    PRINTER_STATES.DataReady :                        // Wait for command to begin printing
                                                    IF NOT printerDataReady THEN
														state := PRINTER_STATES.Idle;
													END_IF
													IF _mode = DEVICE_MODES.Auto AND _amPrintNow THEN
                                                        state := PRINTER_STATES.BeginPrintCycle;
                                                        _amPrintNow := FALSE;
														printHeadDebounce.IN := TRUE;
                                                        oLowerPrintHead := TRUE;
                                                        oRunPrinterRibbonUnwindMotor := TRUE;
														//oPrinterStartPrint := TRUE;
                                                    END_IF                                    
            
    
    PRINTER_STATES.BeginPrintCycle :                // Start printing
                                                    
                                                    
                                                    IF _amSendPrintSignal THEN
                                                        oPrinterStartPrint := TRUE;
														
                                                        state := PRINTER_STATES.Printing;
                                                        printHeadDebounce.IN := FALSE;
                                                        _amSendPrintSignal := FALSE;
                                                    END_IF                                                    
                                        
    
    PRINTER_STATES.FeedAtPrintSpeed :                //

                                                    
                                                                                                
                                        
    PRINTER_STATES.Printing :                        //While printing, wait for End of Print signal
													printerRibbonMovingTimer1.IN := ribbonEncoderPulse;
													printerRibbonMovingTimer2.IN := NOT ribbonEncoderPulse;
                                                    IF endOfPrintONS.Q OR printerRibbonMovingTimer1.Q OR printerRibbonMovingTimer2.Q THEN
                                                        oPrinterStartPrint := FALSE;
                                                        oLowerPrintHead := FALSE;
														IF printerRibbonMovingTimer1.Q OR printerRibbonMovingTimer2.Q THEN
															ribbonFault.Trigger();
														END_IF
														printerRibbonMovingTimer1.IN := FALSE;
														printerRibbonMovingTimer2.IN := FALSE;
														 
                                                        //oRunPrinterRibbonUnwindMotor := FALSE;
                                                        state := PRINTER_STATES.DonePrinting;    
                                                    END_IF
                                        
    PRINTER_STATES.DonePrinting :                    //Done printing, feed a little more through
                                                    IF _mode = DEVICE_MODES.Auto AND _amGoToIdle THEN
                                                        oRunPrinterRibbonUnwindMotor := FALSE;
                                                        state := PRINTER_STATES.Idle;
                                                        _amGoToIdle := FALSE;
														HMIData.printerCycles.Increment();
														HMIData.printHeadClean.Increment();
                                                        Globals.printerCycleCounts := Globals.printerCycleCounts + 1;
                                                    END_IF
        
    PRINTER_STATES.FeedThrough :                        
                                        
    PRINTER_STATES.Ready :                        
                                        
    PRINTER_STATES.Fault :                        
                                        
END_CASE

METHOD AutoSendPrintSignal
VAR_INPUT
END_VAR
_amSendPrintSignal := TRUE;
END_METHOD

METHOD AutoPrintNow
VAR_INPUT
END_VAR
_amPrintNow := TRUE;
END_METHOD

METHOD AutoAckPrintDone
VAR_INPUT
END_VAR
_amGoToIdle := TRUE;
END_METHOD

PROPERTY Ready : BOOL
SET
_ready := Ready;
END_SET
GET
Ready := _ready;
END_GET
END_PROPERTY

PROPERTY Mode : DEVICE_MODES
SET
_mode := Mode;
END_SET
GET
Mode := _mode;
END_GET
END_PROPERTY

END_FUNCTION_BLOCK

// Device/Application/FBs/Components/MonostableMultivibratorFB
FUNCTION_BLOCK MonostableMultivibratorFB EXTENDS BaseComponentFB
VAR_INPUT
END_VAR
VAR_OUTPUT
	Q : BOOL;   // Output pulse
END_VAR
VAR
	_trigger : BOOL;
	_dwellTimeInMS : UINT := 80; 	// Pulse Dwell in mS 
	_delayTimeInMS : UINT; 			// Delay before Pulse in mS
	_manualOn : BOOL;
	_manualOff : BOOL;
	active : BOOL;
	dwellTimer : Standard.TON;
	delayTimer : Standard.TON;
END_VAR


// HPA is on for only as long as its setpoint.

delayTimer(IN := _trigger AND NOT dwellTimer.Q, PT := UINT_TO_TIME(_delayTimeInMS));
dwellTimer(IN := delayTimer.Q AND NOT dwellTimer.Q, PT := UINT_TO_TIME(_dwellTimeInMS));

Q:= delayTimer.Q OR _manualOn;

IF dwellTimer.Q OR _reset THEN
	active := FALSE;
	_trigger := FALSE;
	_manualOn := FALSE;
	_manualOff := FALSE;
END_IF

SUPER^();

PROPERTY DelaySetting : UINT
GET
DelaySetting := _delayTimeInMS;
END_GET
SET
_delayTimeInMS := DelaySetting;
END_SET
END_PROPERTY

METHOD Trigger
VAR_INPUT
END_VAR
_trigger := TRUE;
END_METHOD

METHOD ManualOn
VAR_INPUT
END_VAR
_manualOn := TRUE;
_manualOff := FALSE;
END_METHOD

METHOD ManualOff : BOOL
VAR_INPUT
END_VAR
_manualOn := FALSE;
_manualOff := TRUE;
END_METHOD

PROPERTY DwellSetting : UINT
SET
_dwellTimeInMS := DwellSetting;
END_SET
GET
DwellSetting := _dwellTimeInMS;
END_GET
END_PROPERTY

END_FUNCTION_BLOCK

// Device/Application/FBs/Components/DelayDwellFB/DelayDwellFB
FUNCTION_BLOCK DelayDwellFB EXTENDS BaseComponentFB
VAR_INPUT
END_VAR
VAR_OUTPUT
	Q : BOOL;   // Output pulse
END_VAR
VAR
	_trigger : BOOL;
	_dwellTimeInMS : DINT := 80; 	// Pulse Dwell in mS 
	_delayTimeInMS : DINT; 			// Delay before Pulse in mS
	_manualOn : BOOL;
	_manualOff : BOOL;
	active : BOOL;
	dwellTimer : Standard.TON;
	delayTimer : Standard.TON;
	state : DELAY_DWELL_STATES;
END_VAR

//    Function Block: DelayDwellFB
//    Description: On Trigger(), starts a delay then sets the Q output for a dwell time.  Each addition Trigger() resets the dwell timer.
//    Created by: Ben Hess
//    Created Date: February 20th, 2020

// Setup timers for reading offset and scanning distance
delayTimer(PT := UDINT_TO_TIME(_delayTimeInMS));
// If negative dwell time, run forever
IF _dwellTimeInMS < 0 THEN
	dwellTimer(PT := T#0MS);
ELSE
	dwellTimer(PT := UDINT_TO_TIME(_dwellTimeInMS));
END_IF

// Manual On/Off
IF _manualOff THEN
	THIS^.Reset();
	state := DELAY_DWELL_STATES.Idle;
ELSIF _manualOn THEN
	THIS^.Reset();
	Q := TRUE;
	state := DELAY_DWELL_STATES.Idle;
END_IF

CASE state OF
	DELAY_DWELL_STATES.Idle:  			//
										dwellTimer.IN := FALSE;
										delayTimer.IN := FALSE;
										
										IF _trigger THEN
											IF _delayTimeInMS <> 0 THEN
												state := DELAY_DWELL_STATES.Delay;
											ELSE
												state := DELAY_DWELL_STATES.Dwell;
											END_IF
											_trigger := FALSE;
										END_IF
	
	DELAY_DWELL_STATES.Delay: 			//
										delayTimer.IN := TRUE;
										IF delayTimer.Q THEN
											delayTimer.IN := FALSE;
											state := DELAY_DWELL_STATES.Dwell;
										END_IF
	
	DELAY_DWELL_STATES.Dwell: 			//
										Q := TRUE;
										IF _dwellTimeInMS >= 0 THEN
											dwellTimer.IN := TRUE;
											IF dwellTimer.Q THEN
												dwellTimer.IN := FALSE;
												Q := FALSE;
												state := DELAY_DWELL_STATES.Idle;
											END_IF
										END_IF
										IF _trigger THEN
											_trigger := FALSE;
											state := DELAY_DWELL_STATES.ResettingDwell;
										END_IF
										
	DELAY_DWELL_STATES.ResettingDwell: 	//
										dwellTimer.IN := FALSE;
										state := DELAY_DWELL_STATES.Dwell;
END_CASE

SUPER^();

METHOD Reset : BOOL
VAR_INPUT
END_VAR
active := FALSE;
_trigger := FALSE;
_manualOn := FALSE;
_manualOff := FALSE;
Q := FALSE;
state := DELAY_DWELL_STATES.Idle;
END_METHOD

METHOD ManualOff : BOOL
VAR_INPUT
END_VAR
_manualOn := FALSE;
_manualOff := TRUE;
END_METHOD

METHOD ManualOn
VAR_INPUT
END_VAR
_manualOn := TRUE;
_manualOff := FALSE;
END_METHOD

METHOD Trigger
VAR_INPUT
END_VAR
_trigger := TRUE;
END_METHOD

PROPERTY DwellSetting : DINT
GET
DwellSetting := _dwellTimeInMS;
END_GET
SET
_dwellTimeInMS := DwellSetting;
END_SET
END_PROPERTY

PROPERTY DelaySetting : DINT
SET
_delayTimeInMS := DelaySetting;
END_SET
GET
DelaySetting := _delayTimeInMS;
END_GET
END_PROPERTY

END_FUNCTION_BLOCK

// Device/Application/FBs/Components/BagOpenFingersWithSensorsFB
FUNCTION_BLOCK BagOpenFingersWithSensorsFB EXTENDS BagOpenFingersFB
VAR_INPUT
	rightFingerBagPresent : BOOL;
	leftFingerBagPreset : BOOL;
END_VAR
VAR_IN_OUT
	bagFailedToGrabBothFingersCount : UDINT; // Both Fingers failed to grab bag
	bagFailedToGrabRightFingerCount : UDINT; // Right Bag Open Finger Failed to Grab Bag
	bagFailedToGrabLeftFingerCount : UDINT; // Left Bag Open Finger Failed to Grab Bag
	successfulBagOpenCount : UDINT;			// Successful Bag Open Count
END_VAR
VAR_OUTPUT
	
END_VAR

SUPER^();

METHOD CheckIfBagGrabbed : BOOL
VAR_INPUT
	incrementCounters : BOOL; // IF TRUE Incerment bag counters, otherwise just return bag grabbed status
END_VAR
// Returns true if bag grab successful.  Also increments appropriate counters

{warning disable C0371}
// Checking the VAR_IN_OUT reference, leave the current method in case of invalid reference
IF NOT __ISVALIDREF(successfulBagOpenCount) 
	OR NOT __ISVALIDREF(bagFailedToGrabLeftFingerCount)
	OR NOT __ISVALIDREF(bagFailedToGrabRightFingerCount)
	OR NOT __ISVALIDREF(bagFailedToGrabBothFingersCount)
	THEN RETURN;    
END_IF

IF rightFingerBagPresent AND leftFingerBagPreset THEN
	IF incrementCounters THEN
		successfulBagOpenCount := successfulBagOpenCount +1;
	END_IF
	CheckIfBagGrabbed := TRUE;
ELSIF rightFingerBagPresent AND NOT leftFingerBagPreset THEN
	IF incrementCounters THEN
		bagFailedToGrabLeftFingerCount := bagFailedToGrabLeftFingerCount +1 ;
	END_IF
ELSIF NOT rightFingerBagPresent AND leftFingerBagPreset THEN
	IF incrementCounters THEN
		bagFailedToGrabRightFingerCount := bagFailedToGrabRightFingerCount + 1;
	END_IF
ELSE
	IF incrementCounters THEN
		bagFailedToGrabBothFingersCount := bagFailedToGrabBothFingersCount + 1;
	END_IF
END_IF
{warning restore C0371}
END_METHOD

END_FUNCTION_BLOCK

// Device/Application/FBs/Components/BagOpenFingersFB
FUNCTION_BLOCK BagOpenFingersFB EXTENDS BaseComponentFB
VAR_INPUT

END_VAR
VAR_IN_OUT

END_VAR
VAR_OUTPUT
    releaseOutput : BOOL;
	grabOutput : BOOL;
END_VAR
VAR
    _releaseCommand : BOOL;
    _grabCommand : BOOL;
END_VAR

SUPER^();
releaseOutput := _releaseCommand AND enable;
grabOutput := _grabCommand AND enable;

METHOD Release
VAR_INPUT
END_VAR
_releaseCommand := TRUE;
_grabCommand := FALSE;
END_METHOD

METHOD Grab
VAR_INPUT
END_VAR
_releaseCommand := FALSE;
_grabCommand := TRUE;
HMIData.bagOpenFingerCycles.Increment();
END_METHOD

END_FUNCTION_BLOCK

// Device/Application/FBs/Motors/Applied Motion/FB_AppliedMotionStepServoEIPPassthrough
FUNCTION_BLOCK FB_AppliedMotionStepServoEIPPassthrough EXTENDS FB_AppliedMotionStepServoEIPBase
VAR_INPUT
END_VAR
VAR_OUTPUT
END_VAR
VAR
	homingState : JAW_HOMING_STATES;
	homeRequiredONS : R_TRIG;
	timerHomeDelay : TON;
END_VAR

SUPER^();

METHOD HomeNow
_homeNow := TRUE;
END_METHOD

METHOD DoneClamping
VAR_INPUT
END_VAR
sclCommand := 16#434D; // CM Control Mode
parameter1 := 21;
															
commandSuccessful := FALSE;
commands.SendHostCommand := TRUE;
END_METHOD

METHOD AllowClamping
VAR_INPUT
END_VAR
sclCommand := 16#434D; // CM Control Mode
parameter1 := 1;
															
commandSuccessful := FALSE;
commands.SendHostCommand := TRUE;
END_METHOD

//{warning 'add method implementation '}
METHOD Stop
commandSuccessful := FALSE;
commands.StopCrash := TRUE;
END_METHOD

METHOD SetPositionLimit
VAR_INPUT
	positionLimit : DINT;
END_VAR
sclCommand := 16#5046; // PF (Position Fault)
parameter1 := positionLimit;
															
commandSuccessful := FALSE;
commands.SendHostCommand := TRUE;
END_METHOD

METHOD Execute
VAR_INPUT
END_VAR
SUPER^.Execute();
timerHomeDelay();
homeRequiredONS(CLK := homeRequiredIndication);

//IF _reset OR homeRequiredONS.Q THEN
IF _reset THEN
	homingState := JAW_HOMING_STATES.Idle;
	_homeNow := FALSE;
	timerHomeDelay.IN := FALSE;
END_IF

CASE homingState OF
	JAW_HOMING_STATES.Idle:						IF _homeNow THEN
													//IF NOT driveInputs[10].2 THEN
													//	homingState := JAW_HOMING_STATES.MoveForwardFromSensor;
													//ELSE 
														homingState := JAW_HOMING_STATES.StartHoming;
													//END_IF
													_homeNow := FALSE;
												END_IF
												
	JAW_HOMING_STATES.MoveForwardFromSensor:	commandSuccessful := FALSE;
												velocitySetpoint := 2583;
												pointToPointAccelSetpoint := 1000;
												pointToPointDecelSetpoint := 1000;
												distanceToMoveInSteps := -4000;
												commands.FeedToLength := TRUE;
												homingState := JAW_HOMING_STATES.MovingForwardFromSensor;
												
	JAW_HOMING_STATES.MovingForwardFromSensor:	timerHomeDelay.PT := T#200MS;
												timerHomeDelay.IN := TRUE;
												IF timerHomeDelay.Q THEN
													IF (NOT Moving AND InPosition) THEN
														homingState := JAW_HOMING_STATES.StartHoming;
														timerHomeDelay.IN := FALSE;
                                                       END_IF
												END_IF
												
	JAW_HOMING_STATES.StartHoming:				commandSuccessful := FALSE;
												velocitySetpoint := 1250;
												pointToPointAccelSetpoint := 10;
												pointToPointDecelSetpoint := 10;
												distanceToMoveInSteps := 1;
												ExecuteStoredProgram(2);
												homingState := JAW_HOMING_STATES.Homing;
												
	JAW_HOMING_STATES.Homing:					timerHomeDelay.PT := T#200MS;
												timerHomeDelay.IN := TRUE;
												IF timerHomeDelay.Q THEN
													IF (NOT SUPER^.Homing) THEN
														homingState := JAW_HOMING_STATES.HomeComplete;
														timerHomeDelay.IN := FALSE;
                                                       END_IF
												END_IF 
												
	JAW_HOMING_STATES.HomeComplete:				//MoveToPosition(2, 1000,1000,2583);
												homingState := JAW_HOMING_STATES.SetLimits;

	JAW_HOMING_STATES.MovingToTwoInches : 		timerHomeDelay.PT := T#200MS;
												timerHomeDelay.IN := TRUE;
												IF timerHomeDelay.Q THEN
													IF (NOT Moving AND InPosition) THEN
														homingState := JAW_HOMING_STATES.SetLimits;
														timerHomeDelay.IN := FALSE;
                                                       END_IF
												END_IF 
												
	JAW_HOMING_STATES.SetLimits :				commandSuccessful := FALSE;
												ExecuteStoredProgram(3);
												homingState := JAW_HOMING_STATES.Idle;
												
	
END_CASE
END_METHOD

END_FUNCTION_BLOCK

// Device/Application/FBs/Components/AdjustablePassthroughFB
FUNCTION_BLOCK AdjustablePassthroughFB EXTENDS BaseComponentFB IMPLEMENTS IComponentStatus
VAR_INPUT
	pressureBarEndStopMotor : IPositionableMotor;
	jogInPB : BOOL;
	jogOutPB : BOOL;
END_VAR
VAR_OUTPUT
    homeRequired : BOOL; //Homing Required
    passthroughPosition : REAL;
    state : PASSTHROUGH_SERVO_STATES := PASSTHROUGH_SERVO_STATES.Idle; //State indication of Jaw Passthrough Servo
    exhaustPressureBarRequest : BOOL; // Exhaust pressure bar request for passthrough movement
    extendPressureBarRequest : BOOL; // Extend pressure bar request for passthrough movement
END_VAR
VAR        
    passthroughSetpoint : REAL;        // Passthrough setpoint in inches
	passthroughTravel : REAL;				// Passthrough travel total
	capturePassthroughPos : REAL;
    mustMovePassthroughOut : BOOL; //Flag to tell us that the setpoint requires us to move the passthrough out
    _homeEndStop : BOOL;            // Home End Stop Command
    _movePassthrough  : BOOL;        // Move Passthrough
    _ackRequest : BOOL;                // Request Acknowledged from controller
	passthroughSettingLast : REAL;
	timerHomeDelay : TON;
	faultONS : FB_ONS;
	jogInONS : FB_ONS;
	jogOutONS : FB_ONS;
	
END_VAR
VAR_IN_OUT
	cumulativeChangeCount : DINT;
	cumulativeChangeDistance : UDINT;
END_VAR

//    Function Block: AdjustablePassthroughFB
//    Description:      The adjustable passthrough on the pneumatic head uses a closed loop stepper motor to 
//                    move the end stop for the jaw cylinders
//    Created by: Ben Hess
//    Created Date: Thursday, May 10, 2018
SUPER^();
jogInONS(CLK := jogInPB);
jogOutONS(CLK := jogOutPB);
//Add 2 inch offset
passthroughPosition :=  (pressureBarEndStopMotor.CurrentPosition) - HMIData.passthroughOffset;
timerHomeDelay();
faultONS(CLK := HMIData.faultActive);


//Go to idle when enabled
enableONS(CLK := enable);
IF enableONS.Q OR resetONS.Q THEN    
    state := PASSTHROUGH_SERVO_STATES.Idle;
	_movePassthrough := FALSE;
	Globals.jawMovingIn := FALSE;
	 _homeEndStop := FALSE;
	 timerHomeDelay.IN := FALSE;
	passthroughSetpoint := HMIData.passthroughSetting + HMIData.passthroughOffset ;
END_IF

IF NOT enable THEN
    state := PASSTHROUGH_SERVO_STATES.Idle;
	_movePassthrough := FALSE;
	_homeEndStop := FALSE;
END_IF

_ready := (_mode = DEVICE_MODES.Auto) AND NOT (state = PASSTHROUGH_SERVO_STATES.Fault);
IF faultONS.OSR THEN
	pressureBarEndStopMotor.Stop();
	state := PASSTHROUGH_SERVO_STATES.Idle;
END_IF

CASE state OF
    PASSTHROUGH_SERVO_STATES.Idle :                     // Go to ready state if no home required.  Otherwise go to ready if enabled. Stay in Idle if disabled.
                                                        extendPressureBarRequest := FALSE;
                                                        exhaustPressureBarRequest := FALSE;
														timerHomeDelay.IN := FALSE;
                                                        IF enable AND pressureBarEndStopMotor.HomeRequired THEN
                                                            state := PASSTHROUGH_SERVO_STATES.HomingRequired;
                                                        ELSIF enable THEN
                                                            state := PASSTHROUGH_SERVO_STATES.Ready;
                                                        END_IF
                                                        
    PASSTHROUGH_SERVO_STATES.HomingRequired :            //When Home Servo Pushbitton is pressed
														homeRequired := TRUE;
                                                        IF _homeEndStop THEN
                                                            state := PASSTHROUGH_SERVO_STATES.StartHoming;
                                                        END_IF
                                                        
    PASSTHROUGH_SERVO_STATES.StartHoming :                
                                                        // Start motor homing sequence
                                                        exhaustPressureBarRequest := TRUE;
														Globals.jawMovingIn := TRUE;
														//extendPressureBarRequest := TRUE;
                                                        IF _ackRequest THEN
															pressureBarEndStopMotor.HomeNow();
                                                            exhaustPressureBarRequest := FALSE;
															//extendPressureBarRequest := FALSE;
                                                            _ackRequest := FALSE;
                                                            state := PASSTHROUGH_SERVO_STATES.Homing;    
                                                        END_IF        

    
    PASSTHROUGH_SERVO_STATES.Homing :                    //Move on to Home Complete once finished
														
														timerHomeDelay.PT := T#200MS;
														timerHomeDelay.IN := TRUE;
														IF NOT iPassthroughHomeSensorClear THEN
															extendPressureBarRequest := TRUE;
															Globals.jawMovingIn := FALSE;
														END_IF
														
														IF _ackRequest THEN 
															extendPressureBarRequest := FALSE;
														END_IF 
														
														IF timerHomeDelay.Q THEN
															IF (NOT pressureBarEndStopMotor.HomeRequired) THEN
																state := PASSTHROUGH_SERVO_STATES.HomeComplete;
																extendPressureBarRequest := FALSE;
																_ackRequest := FALSE;
																timerHomeDelay.IN := FALSE;
                                                        	END_IF
														END_IF
                                                        
    
    PASSTHROUGH_SERVO_STATES.HomeComplete :             //Move on to Ready State once supervisor acks the cylinder request
                                                        _homeEndStop := FALSE;
														Globals.jawMovingIn := FALSE;
                                                        extendPressureBarRequest := TRUE;
														homeRequired := FALSE;
                                                        IF _ackRequest THEN
                                                            extendPressureBarRequest := FALSE;
                                                            _ackRequest := FALSE;
                                                            state := PASSTHROUGH_SERVO_STATES.Ready;    
                                                        END_IF
                                                        
    PASSTHROUGH_SERVO_STATES.MovePassthroughOut :        // Move passthrough out
                                                        extendPressureBarRequest := TRUE;
                                                        IF _ackRequest THEN
                                                            pressureBarEndStopMotor.MoveToPosition(position := (passthroughSetpoint + HMIData.passthroughOffset), 
                                                                                    acceleration := 150, 
                                                                                    deceleration := 150, 
                                                                                    velocity := 2583);
                                                            //
                                                            extendPressureBarRequest := FALSE;
                                                            _ackRequest := FALSE;
                                                            state := PASSTHROUGH_SERVO_STATES.MovingPassthroughOut;        
                                                        END_IF
                                                        

                                                    
                                                        
    PASSTHROUGH_SERVO_STATES.MovingPassthroughOut :        //Move on to Passthrough Moved Out once position reached
														timerHomeDelay.PT := T#200MS;
														timerHomeDelay.IN := TRUE;
														IF timerHomeDelay.Q THEN
															IF (REAL_TO_INT((passthroughSetpoint + HMIData.passthroughOffset)*100) = REAL_TO_INT(passthroughPosition*100)) THEN
																state := PASSTHROUGH_SERVO_STATES.PassthroughMovedOut;
																timerHomeDelay.IN := FALSE;
															END_IF
															
															IF jogOutONS.OSF THEN
																passthroughTravel := ABS(capturePassthroughPos - passthroughPosition);
																pressureBarEndStopMotor.Stop();
																Globals.passthroughChangedFromJog := TRUE;
																state := PASSTHROUGH_SERVO_STATES.PassthroughMovedOut;
															END_IF
														END_IF
    PASSTHROUGH_SERVO_STATES.PassthroughMovedOut :       
														extendPressureBarRequest := TRUE; 
                                                         IF _ackRequest THEN
                                                            extendPressureBarRequest := FALSE;
                                                            _movePassthrough := FALSE;
                                                            _ackRequest := FALSE;
															HMIData.passthroughChanges.Increment();
                                                            cumulativeChangeCount := cumulativeChangeCount + 1;
															cumulativeChangeDistance := cumulativeChangeDistance + REAL_TO_UDINT((passthroughTravel * 10));
                                                            state := PASSTHROUGH_SERVO_STATES.Ready;    
                                                        END_IF
                                                        
    PASSTHROUGH_SERVO_STATES.MovePassthroughIn :        
                                                        exhaustPressureBarRequest := TRUE;
														Globals.jawMovingIn := TRUE;
                                                        IF _ackRequest THEN
                                                            pressureBarEndStopMotor.MoveToPosition(position := (passthroughSetpoint + HMIData.passthroughOffset), 
                                                                                    acceleration := 150, 
                                                                                    deceleration := 150, 
                                                                                    velocity := 2583);
                                                            //
                                                            exhaustPressureBarRequest := FALSE;
                                                            _ackRequest := FALSE;
                                                            state := PASSTHROUGH_SERVO_STATES.MovingPassthroughIn;        
                                                        END_IF
                                                    
                                                        
    PASSTHROUGH_SERVO_STATES.MovingPassthroughIn :        //Move on to Passthrough Moved In once position reached
														timerHomeDelay.PT := T#200MS;
														timerHomeDelay.IN := TRUE;
														IF timerHomeDelay.Q THEN
															IF (REAL_TO_INT((passthroughSetpoint + HMIData.passthroughOffset)*100) = REAL_TO_INT(passthroughPosition*100)) THEN
																state := PASSTHROUGH_SERVO_STATES.PassthroughMovedIn;
																timerHomeDelay.IN := FALSE;
															END_IF
															
															IF jogInONS.OSF THEN
																passthroughTravel := ABS(capturePassthroughPos - passthroughPosition);
																pressureBarEndStopMotor.Stop();
																Globals.passthroughChangedFromJog := TRUE;
																state := PASSTHROUGH_SERVO_STATES.PassthroughMovedIn;
															END_IF
                                                        END_IF
    PASSTHROUGH_SERVO_STATES.PassthroughMovedIn :        
                                                        extendPressureBarRequest := TRUE;
														Globals.jawMovingIn := FALSE;
                                                        IF _ackRequest THEN
                                                            extendPressureBarRequest := FALSE;
                                                            _movePassthrough := FALSE;
                                                            _ackRequest := FALSE;
															HMIData.passthroughChanges.Increment();
                                                            cumulativeChangeCount := cumulativeChangeCount + 1;
															cumulativeChangeDistance := cumulativeChangeDistance + REAL_TO_UDINT((passthroughTravel * 10));
                                                            state := PASSTHROUGH_SERVO_STATES.Ready;    
                                                        END_IF
                                                        
                                                        
    PASSTHROUGH_SERVO_STATES.Ready :                    // Keep track    
                                                        IF jogInPB THEN
															passthroughSetpoint := 2.0 + HMIData.passthroughOffset;
															capturePassthroughPos := passthroughPosition;
															state := PASSTHROUGH_SERVO_STATES.MovePassthroughIn;
														ELSIF jogOutPB THEN
															passthroughSetpoint := 8.0 + HMIData.passthroughOffset;
															capturePassthroughPos := passthroughPosition;
															state := PASSTHROUGH_SERVO_STATES.MovePassthroughOut;
														ELSIF jogInONS.OSF OR jogOutONS.OSF THEN
															Globals.passthroughChangedFromJog := TRUE;
															pressureBarEndStopMotor.Stop();
														END_IF
														
                                                        IF _movePassthrough THEN
															passthroughTravel := ABS(passthroughPosition - (passthroughSetpoint + HMIData.passthroughOffset));
                                                            IF mustMovePassthroughOut THEN
                                                                state := PASSTHROUGH_SERVO_STATES.MovePassthroughOut;
                                                                ELSE state := PASSTHROUGH_SERVO_STATES.MovePassthroughIn;
                                                            END_IF
                                                        END_IF
                                                        IF _homeEndStop THEN
                                                            state := PASSTHROUGH_SERVO_STATES.StartHoming;
                                                        END_IF
    
    PASSTHROUGH_SERVO_STATES.Fault :   					pressureBarEndStopMotor.Stop();        
END_CASE

METHOD MovePassthrough
VAR_INPUT
    PassthroughSetting : REAL;
END_VAR
passthroughSetpoint := PassthroughSetting;
mustMovePassthroughOut := (passthroughSetpoint > passthroughPosition);
_movePassthrough := TRUE;
END_METHOD

PROPERTY Ready : BOOL
GET
Ready := _ready;
END_GET
SET
_ready := Ready;
END_SET
END_PROPERTY

PROPERTY Mode : DEVICE_MODES
GET
Mode := _mode;
END_GET
SET
_mode := Mode;
END_SET
END_PROPERTY

METHOD AckRequest
VAR_INPUT
END_VAR
_ackRequest := TRUE;
END_METHOD

METHOD HomeEndStop
VAR_INPUT
END_VAR
_homeEndStop := TRUE;
END_METHOD

END_FUNCTION_BLOCK

// Device/Application/FBs/Cylinders/FB_CylinderFaults
FUNCTION_BLOCK FB_CylinderFaults
VAR_INPUT
	enable : BOOL;
	extendCommand : BOOL;
	extendedInput : BOOL;
	retractCommand : BOOL;
	retractedInput : BOOL;
	faultTime : TIME := T#2500ms;
END_VAR
VAR_OUTPUT
	failToExtend : BOOL;
	failToRetract : BOOL;
END_VAR
VAR
	extendFaultTimer : Standard.TON;
	retractFaultTimer : Standard.TON;
END_VAR
VAR_IN_OUT
END_VAR

extendFaultTimer(PT := faultTime, Q => failToExtend);
retractFaultTimer(PT := faultTime, Q => failToRetract);
IF enable THEN
	IF extendCommand THEN
		retractFaultTimer.IN := FALSE;
		extendFaultTimer.IN := NOT extendedInput;
	ELSIF retractCommand THEN
		extendFaultTimer.IN := FALSE;
		retractFaultTimer.IN := NOT retractedInput;
	ELSE
		retractFaultTimer.IN := FALSE;
		extendFaultTimer.IN := FALSE;
	END_IF
ELSE
	retractFaultTimer.IN := FALSE;
	extendFaultTimer.IN := FALSE;
END_IF

END_FUNCTION_BLOCK

// Device/Application/FBs/FB_HMILight
FUNCTION_BLOCK FB_HMILight
VAR_INPUT
END_VAR
VAR_OUTPUT
	lightOutput : BOOL;
END_VAR
VAR
	_turnOn : BOOL;
	_blinkFast : BOOL;
	_blinkSlow : BOOL;
	blinker : OSCAT_BASIC.PWM_DC := (F := 1, DC := 0.5);
	slowBlinkSec : REAL := 1;
	fastBlinkSec : REAL := 0.5;
END_VAR

IF _blinkFast THEN
	blinker.F := fastBlinkSec;
ELSIF _blinkSlow THEN 
	blinker.F := slowBlinkSec;
END_IF
	
blinker(F:= , DC:= , Q=> );

lightOutput := _turnOn OR (blinker.Q AND (_blinkFast OR _blinkSlow));

METHOD BlinkSlow
VAR_INPUT
END_VAR
_blinkFast := FALSE;
_blinkSlow := TRUE;
_turnOn := FALSE;
END_METHOD

METHOD BlinkFast
VAR_INPUT
END_VAR
_blinkFast := TRUE;
_blinkSlow := FALSE;
_turnOn := FALSE;
END_METHOD

METHOD TurnOff
VAR_INPUT
END_VAR
_blinkFast := FALSE;
_blinkSlow := FALSE;
_turnOn := FALSE;
END_METHOD

METHOD TurnOn
VAR_INPUT
END_VAR
_blinkFast := FALSE;
_blinkSlow := FALSE;
_turnOn := TRUE;
END_METHOD

END_FUNCTION_BLOCK

// Device/Application/FBs/Components/FillerFB
FUNCTION_BLOCK FillerFB EXTENDS BaseComponentFB IMPLEMENTS IComponentStatus
VAR_INPUT
	fillerTrigger : BOOL;
	activateFiller : BOOL;
	fillerOK : BOOL;
	dropTime : REAL;
END_VAR
VAR_OUTPUT
	state : FILLER_STATES;
	fillerModeActive : BOOL;
	waitingForFiller : BOOL;
	cycleBagRequest : BOOL;
	cycleBaggerToActivateFiller : Warning;
	notReady : FB_Fault(name := 'Not Ready');
END_VAR
VAR
	_baggerCycleInitiated : BOOL;
    _baggerCycledAndReady : BOOL;
	fillerRequestedCycle : BOOL;
	fillerTrigONS : FB_ONS;
	dropTimer : Standard.TON;
END_VAR
	
VAR_IN_OUT
END_VAR

//    Function Block: FillerFB
//    Description: Filler state machine
//    Created by: Ben Hess
//    Created Date: October 16th, 2019
SUPER^();
dropTimer(PT := TO_TIME(dropTime * 1000));
IF resetONS.Q OR HMIData.faultActive OR NOT enable OR NOT activateFiller THEN
	state := FILLER_STATES.Idle;
	fillerRequestedCycle := FALSE;
	cycleBaggerToActivateFiller.active := FALSE;
	waitingForFiller := FALSE;
	cycleBagRequest := FALSE;
	_baggerCycledAndReady := FALSE;
	_baggerCycleInitiated := FALSE;
	dropTimer.IN := FALSE;
END_IF

IF NOT fillerOK AND enable AND activateFiller THEN
	notReady.Trigger();
END_IF

fillerTrigONS(CLK := fillerTrigger);
IF fillerTrigONS.OSR THEN
	fillerRequestedCycle := TRUE;
END_IF

CASE state OF
	FILLER_STATES.Idle :							IF (activateFiller AND enable) AND NOT HMIData.faultActive THEN
														state := FILLER_STATES.CycleBaggerToActiveFiller;
													END_IF
	
	FILLER_STATES.CycleBaggerToActiveFiller :		// Operator must cycle a bag out first to guarentee bag open and ready for filler
													cycleBaggerToActivateFiller.active := TRUE;
													
													IF _baggerCycledAndReady THEN
														cycleBaggerToActivateFiller.active := FALSE;
														_baggerCycledAndReady := FALSE;
														fillerRequestedCycle := FALSE;
														state := FILLER_STATES.WaitingForFiller;
													END_IF
	
	FILLER_STATES.WaitingForFiller :				// Waiting for filler trigger to initiate cycle
													waitingForFiller := TRUE;
													IF fillerRequestedCycle THEN
														waitingForFiller := FALSE;	
														//IF NOT HMIData.baggerInhibited.active THEN
															fillerRequestedCycle := FALSE;
															state := FILLER_STATES.Dropping;	
														//END_IF
													END_IF
													
	FILLER_STATES.Dropping :						// Filler is dropping product
													dropTimer.IN := TRUE;
													IF dropTimer.Q THEN
														IF NOT HMIData.baggerInhibited.active THEN
															dropTimer.IN := FALSE;
															cycleBagRequest := TRUE;
															state := FILLER_STATES.BaggerCycling;	
														END_IF
													END_IF
	
	FILLER_STATES.BaggerCycling :					// Wait for bag to open 
													IF _baggerCycleInitiated THEN
														_baggerCycleInitiated := FALSE;
														cycleBagRequest := FALSE;
													END_IF
													
													IF _baggerCycledAndReady THEN
														_baggerCycledAndReady := FALSE;
														state := FILLER_STATES.WaitingForFiller;
													END_IF
	
	FILLER_STATES.Fault :
	
END_CASE

METHOD BaggerCycledAndReady : BOOL
VAR_INPUT
END_VAR
_baggerCycledAndReady := TRUE;
END_METHOD

PROPERTY Ready : BOOL
SET
_ready := Ready;
END_SET
GET
Ready := _ready;
END_GET
END_PROPERTY

METHOD BaggerCycleInitiated : BOOL
VAR_INPUT
END_VAR
_baggerCycleInitiated := TRUE;
END_METHOD

PROPERTY Mode : DEVICE_MODES
SET
_mode := Mode;
END_SET
GET
Mode := _mode;
END_GET
END_PROPERTY

METHOD Reset : BOOL
VAR_INPUT
END_VAR
SUPER^.Reset();
END_METHOD

END_FUNCTION_BLOCK

// Device/Application/FBs/Components/MurrIOFB
FUNCTION_BLOCK MurrIOFB EXTENDS BaseComponentFB IMPLEMENTS IComponentStatus
VAR_INPUT
	headNodeEnabled : BOOL;
	guardNodeEnabled : BOOL;
	printerNodeEnabled : BOOL;
	dischargeNodeEnabled : BOOL;
	auxIONodeEnabled : BOOL;
	configVersion : CONFIG_VERSIONS;
	ptrMachineOptionsManagementOutputs : POINTER TO BYTE;
	ptrSystemStatusInputs : POINTER TO BYTE;
END_VAR
VAR_OUTPUT
	commFailController : FB_Fault(name := 'Communication Fail - Bus Master to Controller');
	commFailNode : FB_Fault(name := 'Communication Fail - Bus Master to I/O Node');
	configActive : Warning;	// I/O Configuration Active, please wait
	ok : BOOL; 		// I/O Configuration and Communication good
END_VAR
VAR
	systemStatusINT : INT;
	systemStatusState : MURR_SYSTEM_STATES;
	MOMConfigLast : BYTE;
	restartBusnodePulse : MonostableMultivibratorFB;
END_VAR
	
VAR_IN_OUT

END_VAR

//    Function Block: MurrIOFB
//    Description: Alarms, faults, configuration of the Murr Cube67+ Bus Node
//    Created by: Ben Hess
//    Created Date: October 16th, 2019
SUPER^();

// Set bit 33 to true for 1 second to reset nodes
restartBusnodePulse.DwellSetting := 1000;
restartBusnodePulse(Q => ptrMachineOptionsManagementOutputs[4].1);

// Exit this FB if invaild pointers set
IF ptrMachineOptionsManagementOutputs = 0 OR ptrSystemStatusInputs = 0 THEN
	RETURN;
END_IF

// MOM config - MOM bits are counted from Slot 001 to 4xx and are counted based on the "Maximium" configuration hard coded in the bus master
// Here we can select which verison of code we have in order to utilize MOM correctly if we add additional modules in the future.
CASE configVersion OF
	CONFIG_VERSIONS.V_1_1 :		//
									ptrMachineOptionsManagementOutputs[0].0 := NOT headNodeEnabled;
									ptrMachineOptionsManagementOutputs[0].1 := NOT guardNodeEnabled;
									ptrMachineOptionsManagementOutputs[0].2 := NOT dischargeNodeEnabled;
									ptrMachineOptionsManagementOutputs[0].3 := NOT printerNodeEnabled;
									ptrMachineOptionsManagementOutputs[0].4 := FALSE;
									
								

	CONFIG_VERSIONS.V_1_2, CONFIG_VERSIONS.V_1_3 : 		// Added aux IO to 1.2 and BCV trigger to 1.3
									ptrMachineOptionsManagementOutputs[0].0 := NOT headNodeEnabled;
									ptrMachineOptionsManagementOutputs[0].1 := NOT guardNodeEnabled;
									ptrMachineOptionsManagementOutputs[0].2 := NOT auxIONodeEnabled;
									ptrMachineOptionsManagementOutputs[0].3 := NOT dischargeNodeEnabled;
									ptrMachineOptionsManagementOutputs[0].4 := NOT printerNodeEnabled;
END_CASE


// Run config if IO bus node is waiting on config
systemStatusINT := ptrSystemStatusInputs^;
systemStatusState := systemStatusINT;

// Prevent a IO node reset on boot for no reason
IF Globals.firstScan THEN
	MOMConfigLast := ptrMachineOptionsManagementOutputs[0];
END_IF

// Trigger fault for node not present, or node seen where one shouldn't be 
IF systemStatusState = MURR_SYSTEM_STATES.No_Comm_To_Configured_Node THEN
	commFailNode.Trigger();
END_IF

// A 0 at system state indicates comm fail to controller
IF systemStatusState = 0 THEN
	commFailController.Trigger();
END_IF

// Alert user to MOM config active
IF systemStatusState = MURR_SYSTEM_STATES.Waiting_For_MOM OR
	systemStatusState = MURR_SYSTEM_STATES.Configuring_MOM OR
	systemStatusState = MURR_SYSTEM_STATES.Internal_Comm_Disabled
THEN
	configActive.active := TRUE;
ELSE
	configActive.active := FALSE;
END_IF

// I/O Block is OK only in this state, otherwise we can't trust any I/O coming back
ok := (systemStatusState = MURR_SYSTEM_STATES.Internal_Comm_OK);

CASE systemStatusState OF

	
	MURR_SYSTEM_STATES.Waiting_For_MOM: 			// Bit 32 is Configure MOM bit
													ptrMachineOptionsManagementOutputs[4].0 := TRUE;
													ptrMachineOptionsManagementOutputs[4].1 := FALSE;
													
	
	MURR_SYSTEM_STATES.Configuring_MOM : 			//
													ptrMachineOptionsManagementOutputs[4].0 := FALSE;
													
											

														
											
ELSE
													ptrMachineOptionsManagementOutputs[4].0 := FALSE;
													//IF config changes here, send it down after restarting
													IF ptrMachineOptionsManagementOutputs[0] <> MOMConfigLast THEN
														restartBusnodePulse.Trigger();
														MOMConfigLast := ptrMachineOptionsManagementOutputs[0];
													END_IF
END_CASE

PROPERTY Mode : DEVICE_MODES
GET
Mode := _mode;
END_GET
SET
_mode := Mode;
END_SET
END_PROPERTY

PROPERTY Ready : BOOL
GET
Ready := _ready;
END_GET
SET
_ready := Ready;
END_SET
END_PROPERTY

END_FUNCTION_BLOCK

// Device/Application/FBs/Components/FunnelFB
FUNCTION_BLOCK FunnelFB EXTENDS BaseComponentFB
VAR_INPUT
	sensorsInstalled : BOOL;							// Are open/closed sensors installed?
	openSensor : BOOL;									// Open sensor input
	closedSensor : BOOL;								// Closed sensor input
END_VAR	
VAR_OUTPUT
	opened : BOOL;										// Funnel Opened status
	closed : BOOL;										// Funnel Closed status
	closeOutput : BOOL;									// Map to physical close output
	openOutput : BOOL;									// Map to physical open output
	failToOpen : FB_Fault(name := 'Failed to Open');	// Failed to Open fault
	failToClose : FB_Fault(name := 'Failed to Close');	// Failed to Close fault
END_VAR
VAR
	_delayTimeInMS : UINT; 								// Delay before open in mS
	_closeReq : BOOL;									// Close reqested from CloseNow()
	_openReq : BOOL;									// Open requested from OpenNow()
	openDelayTimer : Standard.TON;						// Open delay timer
	openingTimer : Standard.TON;						// Opening timer
	closingTimer : Standard.TON;						// Closing timer
	faultTimer : FB_CylinderFaults;						// Fault timer for open/close faults
END_VAR

//    Function Block: FunnelFB
//    Description: Funnel
//    Created by: Ben Hess
//    Created Date: November 18th, 2019

IF _reset THEN
	_openReq := FALSE;
	_closeReq := FALSE;
	openingTimer.IN := FALSE;
	closingTimer.IN := FALSE;
	openDelayTimer.IN := FALSE;
END_IF

// Setup timers
openDelayTimer();
openingTimer();
closingTimer();

// Use opening/closing timers for debounce if sensors enabled
// or for actual opening/closing time after command to move if disabled
IF sensorsInstalled THEN
	openingTimer.IN := openSensor;
	closingTimer.IN := closedSensor;
ELSE
	openingTimer.IN := openOutput;
	closingTimer.IN := closeOutput;
END_IF

// Set open/closed status of funnel
opened := openingTimer.Q;
closed := closingTimer.Q;


// Set physical outputs depending on command
IF enable THEN
	IF _closeReq THEN
		closeOutput := TRUE;
		openOutput := FALSE;
		_closeReq := FALSE;
	ELSIF _openReq THEN
		openDelayTimer.IN := TRUE;
		closeOutput := FALSE;
		openOutput := openDelayTimer.Q;
		_openReq := FALSE;
	END_IF
ELSE
	// Turn everything off if disabled
	closeOutput := FALSE;
	openOutput := FALSE;
	_openReq := FALSE;
	_closeReq := FALSE;
	openingTimer.IN := FALSE;
	closingTimer.IN := FALSE;
	openDelayTimer.IN := FALSE;
END_IF

// Fault timer for failed to reach open/closed sensors
faultTimer(
	enable:= THIS^.enable AND sensorsInstalled, 
	extendCommand:= closeOutput, 
	extendedInput:= closedSensor, 
	retractCommand:= openOutput, 
	retractedInput:= openSensor, 
	faultTime:= T#1S, 
	failToExtend=> failToClose.faultTrigger, 
	failToRetract=> failToOpen.faultTrigger);
	
SUPER^();

PROPERTY DelaySetting : REAL
GET
DelaySetting := TO_REAL(openDelayTimer.PT ) / 1000;
END_GET
SET
openDelayTimer.PT := TO_TIME(DelaySetting * 1000);
END_SET
END_PROPERTY

METHOD CloseNow : BOOL
VAR_INPUT
END_VAR
_closeReq := TRUE;
END_METHOD

PROPERTY OpeningTime : REAL
SET
openingTimer.PT := TO_TIME(OpeningTime * 1000);
END_SET
GET
OpeningTime := TO_REAL(openingTimer.PT) / 1000;
END_GET
END_PROPERTY

METHOD OpenNow : BOOL
VAR_INPUT
END_VAR
_openReq := TRUE;
END_METHOD

PROPERTY ClosingTime : REAL
GET
ClosingTime := TO_REAL(closingTimer.PT) / 1000;
END_GET
SET
closingTimer.PT := TO_TIME(ClosingTime * 1000);
END_SET
END_PROPERTY

END_FUNCTION_BLOCK

// Device/Application/FBs/Components/BarcodeReaderFB
FUNCTION_BLOCK BarcodeReaderFB EXTENDS BaseComponentFB
VAR_INPUT
	feedSpeed : REAL;
	positionOffset : REAL;
	distanceToScan : REAL;
	readGoodInput : BOOL;
	badReadFaultCountSetting : UDINT;
END_VAR	
VAR_OUTPUT
	triggerScannerOutput : BOOL;
	xBusy : BOOL;
	xDone : BOOL;
	currentGoodReadCount : UDINT;
	currentBadReadCount : UDINT;
	barcodeFault : BOOL;
END_VAR
VAR
	_goodRead : BOOL;
	_badread : BOOL;
	_trigger : BOOL;
	state : BCR_STATES;
	waitForReadTimer : Standard.TON;
	positionOffsetDelay : Standard.TON;
END_VAR
VAR CONSTANT
	MILLISECONDS_IN_SECOND : INT := 1000;
END_VAR

//    Function Block: BarcodeReaderFB
//    Description: Trigger the barcode verifier and receive a "Barcode OK" signal, or nothing which indicates no read.
//    Created by: Ben Hess
//    Created Date: January 29th, 2020

// Setup timers for reading offset and scanning distance
IF positionOffset > 0 THEN
	positionOffsetDelay(PT := TO_TIME(MILLISECONDS_IN_SECOND / (feedSpeed / positionOffset)) + T#120ms);
ELSE
	positionOffsetDelay(PT := T#0S);
END_IF

IF distanceToScan > 0 THEN
	waitForReadTimer(PT := TO_TIME(MILLISECONDS_IN_SECOND / (feedSpeed / distanceToScan)));
ELSE
	waitForReadTimer(PT := T#0S);
END_IF

IF _reset OR NOT enable THEN
	//
	state := BCR_STATES.Idle;
	barcodeFault := FALSE;
END_IF

CASE state OF
	
	BCR_STATES.Idle:				// Wait for trigger
									triggerScannerOutput := FALSE;
									waitForReadTimer.IN := FALSE;
									positionOffsetDelay.IN := FALSE;
									
									xBusy := FALSE;
									IF _trigger THEN
										state := BCR_STATES.WaitForOffset;
										positionOffsetDelay.IN := TRUE;
										xBusy := TRUE;
										xDone := FALSE;
									END_IF
									
									_trigger := FALSE;
									
	BCR_STATES.WaitForOffset: 		// Wait for offset to trigger read
									IF positionOffsetDelay.Q THEN
										state := BCR_STATES.TriggerReader;
										positionOffsetDelay.IN := FALSE;
									END_IF
									
	BCR_STATES.TriggerReader:		// Trigger the reader and then move to waiting state for result
									triggerScannerOutput := TRUE;
									waitForReadTimer.IN := TRUE;
									state := BCR_STATES.WaitingForResult;
									
	
	BCR_STATES.WaitingForResult:	// Wait for delayToCheckReadStatus timer.  If it times out we did not get a good read
									IF readGoodInput THEN
										_goodRead := TRUE;
										_badread := FALSE;
										currentGoodReadCount := currentGoodReadCount + 1;
										currentBadReadCount := 0;
										xDone := TRUE;
										state := BCR_STATES.Idle;
									ELSIF waitForReadTimer.Q THEN
										_goodRead := FALSE;
										_badread := TRUE;
										currentGoodReadCount := 0;
										currentBadReadCount := currentBadReadCount + 1;
										IF badReadFaultCountSetting > 0 THEN
											IF currentBadReadCount >= badReadFaultCountSetting THEN
												barcodeFault := TRUE;
											END_IF
										END_IF
										xDone := TRUE;
										state := BCR_STATES.Idle;
									END_IF
	
	BCR_STATES.Resetting:
	
END_CASE

SUPER^();

METHOD Trigger : BOOL
VAR_INPUT
END_VAR
_trigger := TRUE;
END_METHOD

PROPERTY BadRead : BOOL
SET
END_SET
GET
END_GET
END_PROPERTY

PROPERTY GoodRead : BOOL
GET
END_GET
SET
END_SET
END_PROPERTY

END_FUNCTION_BLOCK

// Device/Application/FBs/Components/KeyenceL20FB/KeyenceNL20FB
FUNCTION_BLOCK KeyenceNL20FB EXTENDS BaseComponentFB IMPLEMENTS IComponentStatus
VAR_INPUT
	ptrEIPInputs : POINTER TO WORD;
	ptrEIPOutputs : POINTER TO WORD;
	triggerInput : BOOL;
END_VAR
VAR_OUTPUT
	commFail : FB_Fault(name := 'Communication Fail - Bus Master to Controller');
	lastReadData : STRING[100];
	xBusy : BOOL;
	xDone : BOOL;
	goodRead : BOOL;
	badRead : BOOL;
END_VAR
VAR
	error : BOOL;
	readDataUpdateAvailable : BOOL;
	readDataUpdateComplete : BOOL;
	bufferOverflowError : BOOL;
	generalError : BOOL;
	bcvBusy : BOOL;
	readingComplete : BOOL;
	in1Status : BOOL;
	in2Status : BOOL;
	out1Status : BOOL;
	out2Status : BOOL;
	out3Status : BOOL;
	out4Status : BOOL;
	errorCode : UINT;
	readDataReadyCount : UINT;
	readDataUpdateCount : UINT;
	readDataLength : UINT;
	readData : POINTER TO STRING[100];
	
	readDataUpdatePermitted : BOOL;
	errorAndBufferClear : BOOL;
	readingStartRequest : BOOL;
	readingCompleteAck : BOOL;
	bankNumber : UINT;
	
	state : eKeyenceLN20FB_States;
	triggerONS : FB_ONS;
END_VAR
	
VAR_IN_OUT

END_VAR

//    Function Block: KeyenceL20FB
//    Description: Alarms, faults, configuration of the Keyence L-N20 barcode scanner base
//    Created by: Ben Hess
//    Created Date: Feb 28th, 2020


// Exit FB if pointers are invalid
IF ptrEIPInputs = 0 OR ptrEIPOutputs = 0 THEN
	RETURN;
END_IF
triggerONS(CLK := triggerInput);
// Map statuses to friendly variables
error := ptrEIPInputs[0].0;
readDataUpdateAvailable := ptrEIPInputs[0].1;
readDataUpdateComplete := ptrEIPInputs[0].2;
bufferOverflowError := ptrEIPInputs[0].6;
generalError := ptrEIPInputs[0].7;
bcvBusy := ptrEIPInputs[0].8;

readingComplete := ptrEIPInputs[1].0;

in1Status := ptrEIPInputs[2].0;
in2Status := ptrEIPInputs[2].1;
out1Status := ptrEIPInputs[2].4;
out2Status := ptrEIPInputs[2].5;
out3Status := ptrEIPInputs[2].6;
out4Status := ptrEIPInputs[2].7;

errorCode := ptrEIPInputs[16];

readDataReadyCount := ptrEIPInputs[18];
readDataUpdateCount := ptrEIPInputs[19];

readDataLength := ptrEIPInputs[21];
readData := ADR(ptrEIPInputs[22]);


IF resetONS.Q THEN
	state := eKeyenceLN20FB_States.Reset;
END_IF



CASE state OF
	eKeyenceLN20FB_States.Idle: 			//
											
											IF triggerONS.OSR THEN
												readingStartRequest := TRUE;
												xBusy := TRUE;
												xDone := FALSE;
												badRead := FALSE;
												goodRead := FALSE;
												lastReadData := '---Read in Progress---';
												state := eKeyenceLN20FB_States.WaitForStatus;
											END_IF

	eKeyenceLN20FB_States.WaitForStatus:	//
											IF readingComplete OR NOT triggerInput THEN
												state := eKeyenceLN20FB_States.SetStatus;
												readingStartRequest := FALSE;
												readingCompleteAck := TRUE;
											END_IF
	
	eKeyenceLN20FB_States.SetStatus:		// Set the current read status and string
											// If trigger input goes away or barcode error seen set bad read
											IF NOT triggerInput OR out2Status THEN
												badRead := TRUE;
												goodRead := FALSE;
												state := eKeyenceLN20FB_States.WaitForReadClear;
												IF out2Status THEN
													lastReadData := '---BAD READ---';
												ELSE
													lastReadData := '---NO READ---';
												END_IF
											ELSIF out1Status THEN
												goodRead := TRUE;
												badRead := FALSE;
												// Strip terminating char (0x0D) from string to get clean read barcode
												lastReadData := LEFT(readData^, readDataLength - 1);
												state := eKeyenceLN20FB_States.WaitForReadClear;
											END_IF
											
	eKeyenceLN20FB_States.WaitForReadClear:	//
											IF NOT readingComplete THEN
												readingCompleteAck := FALSE;
												xBusy := FALSE;
												xDone := TRUE;
												state := eKeyenceLN20FB_States.Idle;
											END_IF 									

	eKeyenceLN20FB_States.Reset: 			//
											IF readingComplete THEN
												readingCompleteAck := TRUE;
												state := eKeyenceLN20FB_States.WaitForReadClear;
											ELSE
												readingStartRequest := FALSE;
												readingCompleteAck := FALSE;
												xBusy := FALSE;
												xDone := FALSE;
												badRead := FALSE;
												goodRead := FALSE;
												state := eKeyenceLN20FB_States.Idle;
											END_IF
END_CASE	

// Outputs to barcode verifier
ptrEIPOutputs[0].1 :=  readDataUpdatePermitted;
ptrEIPOutputs[0].7 :=  errorAndBufferClear;
ptrEIPOutputs[0].8 := readingStartRequest;
ptrEIPOutputs[1].0 := readingCompleteAck;
ptrEIPOutputs[2] := bankNumber;

// Call to super FB.
SUPER^();

PROPERTY Ready : BOOL
SET
_ready := Ready;
END_SET
GET
Ready := _ready;
END_GET
END_PROPERTY

PROPERTY Mode : DEVICE_MODES
SET
_mode := Mode;
END_SET
GET
Mode := _mode;
END_GET
END_PROPERTY

END_FUNCTION_BLOCK

// Device/Application/FBs/Components/FB_MotorizedPressureBar/FB_MotorizedPressureBar
FUNCTION_BLOCK FB_MotorizedPressureBar EXTENDS BaseComponentFB
VAR_INPUT
	iPressureBarClamped: BOOL;
	iPressureBarClosed : BOOL;
	iPressureBarNotObstructed : BOOL;
	iBaggerEnableButton : BOOL;
	iJawClampExtended : BOOL;
	iJawCLampRetracted : BOOL;
	pbarOutSetting : REAL := 12.0;
	pbarInSetting : REAL := 0.03;
	closeDelay : REAL;
	disableFaults : BOOL;
	extendJawClamp : BOOL;
	retractJawClamp : BOOL;
	extendJaw : BOOL;
	retractJaw : BOOL;
END_VAR
VAR_OUTPUT
	
	
	failToClampLeft : FB_Fault(name := 'Pbar Left Fail to Clamp');
	failToReleaseLeft : FB_Fault(name := 'Pbar Left Fail to Release');
	failToClampRight : FB_Fault(name := 'Pbar Right Fail to Clamp');
	failToReleaseRight : FB_Fault(name := 'Pbar Right Fail to Release');
	faults : PressureBarFaultsType;
	state : MotorizedPbarStates;
	actualPosition : REAL;
	pressureBarOpen : BOOL;
	pressureBarClosed : BOOL;
	homeRequired : BOOL;
	clamped : BOOL;
END_VAR
VAR
	_homeNow : BOOL;
	_openJaw : BOOL;
	_closeJaw : BOOL;
	_closeJawNoLatch : BOOL;
	jawClampsDelay : TIME := T#75ms;
	accel : INT := 40;
	decel : INT := 60;
	velo : INT := 1250;
	testCurrent : DINT := 500;
	testZeroCurrent : BOOL;
	testSomeCurrent : BOOL;
	testClamp : BOOL;
	testRelease : BOOL;
	testPosLimit : BOOL;
	testDisable : BOOL;
	testEnable : BOOL;
	testResetPosition : BOOL;
	posLimit : DINT := 3000;
	pbarFeedbackHandler : FB_CylinderFeedback;
	jawClampsLeftFeedbackHandler : FB_CylinderFeedback;
	jawClampsRightFeedbackHandler : FB_CylinderFeedback;
	startTest : BOOL;
	testActive : BOOL;
	movePassthroughNow : BOOL;
	delayTimer : Standard.TON := (PT:= T#500MS);
	failTimer : Standard.TON := (PT:= T#500MS);
	homeRequiredONS : FB_ONS;
	faultingONS : FB_ONS;
	faultTimeMultiplier : REAL := 150;
	distanceToMove : REAL;
END_VAR
VAR_IN_OUT
	jawClamps : FB_ThreePositionCylinder;
	pbarMotor : FB_AppliedMotionStepServoEIPPassthrough;
	//IBDMotor : FB_AppliedMotionStepServoEIPPassthrough;
END_VAR


actualPosition := pbarMotor.absolutePositonInches;
pressureBarOpen := TO_DINT(actualPosition * 1000) >= (TO_DINT(pbarOutSetting * 1000) - 10) AND TO_DINT(actualPosition * 1000) <= (TO_DINT(pbarOutSetting * 1000) + 10);
//pressureBarClosed := pbarMotor.absolutePositionSteps >= (pbarMotor.distanceToMoveInSteps - 4) AND pbarMotor.absolutePositionSteps <= (pbarMotor.distanceToMoveInSteps + 4);
pressureBarClosed := iPressureBarClosed;
delayTimer();
failTimer(IN := (state = MotorizedPbarStates.StartedClamping) AND (NOT iPressureBarClamped OR NOT iPressureBarClosed));
clamped := state = MotorizedPbarStates.Clamping;





// jawClampsLeftFeedbackHandler(
// 	extendedFeedbackInput:= iJawClampLeftExtended, 
// 	retractedFeedbackInput:= iJawCLampLeftRetracted, 
// 	extendOutput:= jawClamps.extendOutput, 
// 	retractOutput:= jawClamps.retractOutput, 
// 	extendFaultDelay:= 1000, 
// 	retractFaultDelay:= 1000, 
// 	faultMonitoring:= NOT disableFaults, 
// 	failedToExtend=> failToReleaseLeft.faultTrigger, 
// 	failedToRetract=> failToClampLeft.faultTrigger);
// 
// jawClampsRightFeedbackHandler(
// 	extendedFeedbackInput:= iJawClampRightExtended, 
// 	retractedFeedbackInput:= iJawCLampRightRetracted, 
// 	retractOutput:= jawClamps.retractOutput, 
// 	extendOutput:= jawClamps.extendOutput, 
// 	extendFaultDelay:= 1000, 
// 	retractFaultDelay:= 1000, 
// 	faultMonitoring:= NOT disableFaults, 
// 	failedToExtend=> failToReleaseRight.faultTrigger, 
// 	failedToRetract=> failToClampRight.faultTrigger);


IF extendJawClamp THEN
	extendJawClamp := FALSE;
	jawClamps.Extend();
ELSIF retractJawClamp THEN
	retractJawClamp := FALSE;
	jawClamps.Retract();
END_IF

IF NOT pbarMotor.HomeRequired THEN
	IF extendJaw THEN
		extendJaw := FALSE;
		pbarMotor.MoveToPositionTorque(pbarOutSetting,accel,decel,velo,testCurrent);
	ELSIF retractJaw THEN
		retractJaw := FALSE;
		pbarMotor.MoveToPositionTorque(pbarInSetting,accel,decel,velo,testCurrent);
	END_IF
END_IF

IF testDisable THEN
	pbarMotor.Disable();
	testDisable := FALSE;
END_IF

IF testEnable THEN
	pbarMotor.Enable();
	testEnable := FALSE;
END_IF

IF testClamp THEN
	pbarMotor.AllowClamping();
	testClamp := FALSE;
END_IF

IF testRelease THEN
	pbarMotor.DoneClamping();
	testRelease := FALSE;
END_IF

IF testResetPosition THEN
	pbarMotor.ResetEncoderPosition(pbarMotor.driveInputs[5]);
	testResetPosition := FALSE;
END_IF

IF testZeroCurrent THEN
	pbarMotor.MoveDistanceTorque(velocity:=100, acceleration := 1, deceleration := 1, distance := 0, current := 1);
	//pbarMotor.SetTorque(1);
	testZeroCurrent := FALSE;
END_IF

IF testSomeCurrent THEN
	pbarMotor.SetTorque(testCurrent);
	testSomeCurrent := FALSE;
END_IF

IF testPosLimit THEN
	pbarMotor.SetPositionLimit(posLimit);
	testPosLimit := FALSE;
END_IF

IF resetONS.Q THEN
	pbarMotor.Reset();
	//pbarMotor.Enable();
	
	//IBDMotor.Reset();
	Globals.jawMovingIn := FALSE;
	_reset := FALSE;
	startTest := FALSE;
	testActive := FALSE;
	delayTimer.IN := FALSE;
	pbarMotor.DoneClamping();
	jawClamps.Extend();
	pbarFeedbackHandler.extendOutput := FALSE;
	pbarFeedbackHandler.retractOutput := FALSE;
	state := MotorizedPbarStates.Idle; 
END_IF
faultingONS(CLK := (	pbarMotor.Faulted AND NOT disableFaults)
	OR (pbarFeedbackHandler.faultIndication
	OR jawClampsLeftFeedbackHandler.faultIndication
	OR jawClampsRightFeedbackHandler.faultIndication
	OR faults.obstructionDetected.active));

IF 	faultingONS.OSR
	AND state <> MotorizedPbarStates.Faulted 
THEN
	state := MotorizedPbarStates.Faulting; 
END_IF

homeRequiredONS(CLK := pbarMotor.homeRequired);
IF homeRequiredONS.OSR THEN
	homeRequired := TRUE;
END_IF


_ready := state = MotorizedPbarStates.Idle AND NOT homeRequired AND pressureBarOpen;

CASE state OF
	MotorizedPbarStates.Idle :					//
										IF startTest THEN
											startTest := FALSE;
											testActive := TRUE;
											IF pbarMotor.homeRequired THEN
												pbarMotor.HomeNow();
												state := MotorizedPbarStates.Homing;
											ELSE
												state := MotorizedPbarStates.Initialize;
											END_IF
												
										END_IF
											
										IF _homeNow THEN
											_homeNow := FALSE;
											//IF (pbarMotor.homeRequired) THEN
												pbarMotor.HomeNow();
											//END_IF
											delayTimer.PT := T#150MS;
											delayTimer.IN := TRUE;
											state := MotorizedPbarStates.Homing;
										END_IF
										
										IF _openJaw AND NOT _reset THEN
											//pbarMotor.DoneClamping();
											_openJaw := FALSE;
											state := MotorizedPbarStates.MoveJawOut;
										END_IF
										
										IF _closeJaw THEN
											_closeJaw := FALSE;
											state := MotorizedPbarStates.MoveJawIn;
										END_IF
										
										IF _closeJawNoLatch THEN
											//_closeJawNoLatch := FALSE;
											state := MotorizedPbarStates.MoveJawIn;
										END_IF
	
	MotorizedPbarStates.Homing :				//
										Globals.jawMovingIn := TRUE;
										IF NOT (pbarMotor.homeRequired) AND delayTimer.Q THEN
												delayTimer.IN := FALSE;
												//pbarMotor.DoneClamping();
												
												homeRequired := FALSE;
												
												state := MotorizedPbarStates.Initialize;
										END_IF
	
	
	MotorizedPbarStates.Initialize :			//
										delayTimer.PT := T#500MS;
										delayTimer.IN := TRUE;
										Globals.jawMovingIn := TRUE;
										IF delayTimer.Q THEN
											IF pressureBarOpen THEN
												state := MotorizedPbarStates.Initialized;
											ELSE
												jawClamps.Extend();
												pbarMotor.MoveToPositionTorque(pbarOutSetting,accel,decel,velo,testCurrent);
												//IBDMotor.MoveToPosition(pbarOutSetting,accel,decel,velo);
												state := MotorizedPbarStates.Initializing;
											END_IF
											delayTimer.IN := FALSE;
										END_IF
										
	
	
	MotorizedPbarStates.Initializing :			//
										IF pressureBarOpen THEN
											state := MotorizedPbarStates.Initialized;
										END_IF
	
	
	MotorizedPbarStates.Initialized :			//
										IF testActive THEN
											state := MotorizedPbarStates.MoveJawIn;
										ELSE
											state := MotorizedPbarStates.Idle;
										END_IF
										
	
	
	MotorizedPbarStates.MoveJawOut :			//
										
										Globals.jawMovingIn := FALSE;
										pbarMotor.MoveToPositionTorque(pbarOutSetting,accel,decel,velo,testCurrent);
										//IBDMotor.MoveToPosition(pbarOutSetting,accel,decel,velo);
										distanceToMove := ABS(actualPosition - pbarOutSetting);
										state := MotorizedPbarStates.MovingJawOut;
										//pbarMotor.SetPositionLimit(150);
	
	MotorizedPbarStates.MovingJawOut :			//
										IF pressureBarOpen THEN
											
											IF testActive THEN
												delayTimer.PT := T#500MS;
												delayTimer.IN := TRUE;
												IF delayTimer.Q  THEN
													delayTimer.IN := FALSE;
													state := MotorizedPbarStates.MoveJawIn;
												END_IF
											ELSE
												delayTimer.PT := T#100MS;
												delayTimer.IN := TRUE;
												IF delayTimer.Q  THEN
													//pbarMotor.ResetEncoderPosition(pbarMotor.driveInputs[5]);
													delayTimer.IN := FALSE;
													state := MotorizedPbarStates.Idle;
												END_IF
											END_IF
										END_IF
	
	
	MotorizedPbarStates.MovedJawOut :			//
										IF delayTimer.Q THEN
											delayTimer.IN := FALSE;
											state := MotorizedPbarStates.MoveJawIn;
										END_IF
	
	
	MotorizedPbarStates.MoveJawIn :				//
										Globals.jawMovingIn := TRUE;
										pbarMotor.MoveToPositionTorque(pbarInSetting,accel,decel,velo,testCurrent);
										//pbarMotor.MoveToPositionTorque(pbarInSetting,accel,decel,velo,testCurrent);
										//IBDMotor.MoveToPosition(0,accel,decel,velo+(TO_INT(TO_REAL(velo)*0.25)));
										distanceToMove := ABS(actualPosition - pbarInSetting);
										state := MotorizedPbarStates.MovingJawIn;
	
	
	MotorizedPbarStates.MovingJawIn : 			//
										//IF iPressureBarClosed AND pbarMotor.absolutePositonInches = 0 THEN
										IF iPressureBarClosed THEN
											IF NOT  _closeJawNoLatch THEN
												pbarMotor.AllowClamping();
											END_IF
											
											delayTimer.PT := jawClampsDelay;
											delayTimer.IN := TRUE;
											//pbarMotor.Disable();
											state := MotorizedPbarStates.MovedJawIn;
										END_IF
	
	
	MotorizedPbarStates.MovedJawIn :			//
										IF delayTimer.Q THEN
											delayTimer.IN := FALSE;
											IF _closeJawNoLatch THEN
												_closeJawNoLatch := FALSE;
												state := MotorizedPbarStates.Idle;
											ELSE
												state := MotorizedPbarStates.StartClamping;
											END_IF
										END_IF
										
	
	
	MotorizedPbarStates.StartClamping :			//
										//pbarMotor.SetPositionLimit(20000);
										jawClamps.Retract();
										state := MotorizedPbarStates.StartedClamping;
	
	MotorizedPbarStates.StartedClamping :		//
										IF iPressureBarClamped THEN
											delayTimer.PT := T#250MS;
											delayTimer.IN := TRUE;
											IF delayTimer.Q THEN
												pbarMotor.ResetEncoderPosition(pbarMotor.driveInputs[5]);
												state := MotorizedPbarStates.Clamping;	
											END_IF
										END_IF
										
										
										IF testActive THEN
											delayTimer.PT := T#2S;
											delayTimer.IN := TRUE;
										END_IF
	
	
	MotorizedPbarStates.Clamping :				//
										IF _openJaw OR (testActive AND delayTimer.Q) THEN
											_openJaw := FALSE;
											delayTimer.IN := FALSE;
											jawClamps.Extend();
											state := MotorizedPbarStates.ReleaseClamp;
										END_IF
										
	
	
	
	MotorizedPbarStates.ReleaseClamp :			//  
										IF iJawClampExtended THEN
											pbarMotor.DoneClamping();
											//pbarMotor.Enable();
											delayTimer.PT := jawClampsDelay;
											delayTimer.IN := TRUE;
											state := MotorizedPbarStates.ReleasingClamp;
										END_IF
										
	
	
	MotorizedPbarStates.ReleasingClamp :		//
										IF delayTimer.Q THEN
											delayTimer.IN := FALSE;
											state := MotorizedPbarStates.MoveJawOut;
											//HMI.data.TFBeltPressureBarCycles := HMI.data.TFBeltPressureBarCycles + 1;
										END_IF
	
	MotorizedPbarStates.Faulting :			// 
										Globals.jawMovingIn := FALSE;
										_reset := FALSE;
										_openJaw := FALSE;
										_closeJaw := FALSE;
										_homeNow := FALSE;
										_closeJawNoLatch := FALSE;
										startTest := FALSE;
										testActive := FALSE;
										delayTimer.IN := FALSE;
										jawClamps.Extend();
										pbarFeedbackHandler.extendOutput := FALSE;
										pbarFeedbackHandler.retractOutput := FALSE;
										pbarMotor.Disable();
										//IBDMotor.Disable();
										state := MotorizedPbarStates.Faulted;
			
	MotorizedPbarStates.Faulted :				//
	
END_CASE


IF pbarMotor.alarms.positionLimit OR failTimer.Q THEN
	faults.obstructionDetected.Trigger();
	homeRequired := TRUE;
	//state := MotorizedPbarStates.Faulting;
END_IF

pbarFeedbackHandler(
	extendedFeedbackInput:= pressureBarOpen, 
	retractedFeedbackInput:= iPressureBarClosed, 
	extendOutput:= state = MotorizedPbarStates.MovingJawOut, 
	retractOutput:= state = MotorizedPbarStates.MovingJawIn, 
	extendFaultDelay:= TO_INT((distanceToMove) * faultTimeMultiplier) , 
	retractFaultDelay:= TO_INT((distanceToMove) * faultTimeMultiplier), 
	faultMonitoring:= NOT disableFaults, 
	failedToExtend=> faults.failedToOpen.faultTrigger, 
	failedToRetract=> faults.failedToClose.faultTrigger);
	
SUPER^();

METHOD CloseJawNoLatch : BOOL
VAR_INPUT
END_VAR
_closeJawNoLatch := TRUE;
END_METHOD

METHOD CloseJaw : BOOL
VAR_INPUT
END_VAR
_closeJaw := TRUE;
END_METHOD

METHOD OpenJaw : BOOL
VAR_INPUT
END_VAR
_openJaw := TRUE;
END_METHOD

METHOD HomeNow : BOOL
VAR_INPUT
END_VAR
_homeNow := TRUE;
END_METHOD

END_FUNCTION_BLOCK

// Device/Application/FBs/Components/FB_MotorizedPressureBar/FB_CylinderFeedback
FUNCTION_BLOCK FB_CylinderFeedback
VAR_INPUT
    extendedFeedbackInput : BOOL;    //Extended feedback input from I/O
    retractedFeedbackInput : BOOL;    //Retracted feedback input from I/O
	extendOutput : BOOL;				// Extend output from valve
	retractOutput : BOOL; 				// Retract output from valve
    extendFaultDelay : INT := 1000;        //Extend fault delay in MS
    retractFaultDelay : INT := 1000;        //Retract fault delay in MS
    faultMonitoring : BOOL;                    //Fault monitoring enabled if true
END_VAR
VAR_OUTPUT
    failedToExtend : BOOL;            //Failed to Extend Fault
    failedToRetract : BOOL;            //Failed to Retract Fault
	faultIndication : BOOL;            //Overall fault status of cylinder
END_VAR
VAR
    
    extendFaultTimer : TON;            //Extend Fault Timer
    retractFaultTimer : TON;        //Retract Fault Timer
END_VAR

//This code monitors the positon of the cylinder and raises a fault if the cylinder doesn't reach its
//desired postion within the specified time.

//Initialize timers
extendFaultTimer(PT := INT_TO_TIME(extendFaultDelay));
retractFaultTimer(PT := INT_TO_TIME(retractFaultDelay));

//Only enable timers if we are to be monitoring faults
IF faultMonitoring THEN
    extendFaultTimer.IN := (extendOutput AND NOT extendedFeedbackInput);
    retractFaultTimer.IN := (retractOutput AND NOT retractedFeedbackInput);
ELSE 
        extendFaultTimer.IN := FALSE;
        retractFaultTimer.IN := FALSE;
END_IF

//Rasie the alarms
failedToExtend := extendFaultTimer.Q;
failedToRetract := retractFaultTimer.Q;

//Set overall fault indication
faultIndication := failedToExtend OR failedToRetract;

END_FUNCTION_BLOCK

// Device/Application/FBs/Components/FB_MotorizedIBD/FB_MotorizedIBD
FUNCTION_BLOCK FB_MotorizedIBD EXTENDS BaseComponentFB
VAR_INPUT
	pbarOutSetting : REAL := 12.0;
	pbarInSetting : REAL;
	disableFaults : BOOL;
	extendCommand : BOOL;
	retractCommand : BOOL;
END_VAR
VAR_OUTPUT
	
	failToClose : FB_Fault(name := 'IBD Fail to Close');
	failToOpen : FB_Fault(name := 'IBD Fail to Open');
	state : MotorizedIBDStates;
	actualPosition : REAL;
	IBDOpen : BOOL;
	IBDFullyOpen : BOOL;
	homeRequired : BOOL;
	clamped : BOOL;
END_VAR
VAR
	_homeNow : BOOL;
	_openIBD : BOOL;
	_closeIBD : BOOL;
	_openFull : BOOL;
	accel : INT := 100;
	decel : INT := 100;
	velo : INT := 2500;
	testCurrent : DINT := 500;
	testZeroCurrent : BOOL;
	testSomeCurrent : BOOL;
	startTest : BOOL;
	testActive : BOOL;
	movePassthroughNow : BOOL;
	delayTimer : Standard.TON := (PT:= T#500MS);
	homeRequiredONS : FB_ONS;
END_VAR
VAR_IN_OUT
	IBDMotor : FB_AppliedMotionStepServoEIPPassthrough;
END_VAR


actualPosition := IBDMotor.absolutePositonInches;
IBDOpen := TO_DINT(actualPosition * 1000) >= (TO_DINT(pbarOutSetting * 1000) - 10) AND TO_DINT(actualPosition * 1000) <= (TO_DINT(pbarOutSetting * 1000) + 10);
IBDFullyOpen := TO_DINT(actualPosition * 1000) >= (TO_DINT(12 * 1000) - 10) AND TO_DINT(actualPosition * 1000) <= (TO_DINT(12 * 1000) + 10);
//IBDOpen := TO_DINT(IBDMotor.absolutePositonInches) = TO_DINT(pbarOutSetting);
delayTimer();

clamped := state = MotorizedIBDStates.Clamping;


IF NOT IBDMotor.HomeRequired THEN
	IF extendCommand THEN
		extendCommand := FALSE;
		IBDMotor.MoveToPositionTorque(pbarOutSetting,accel,decel,velo,testCurrent);
	ELSIF retractCommand THEN
		retractCommand := FALSE;
		IBDMotor.MoveToPositionTorque(pbarInSetting,accel,decel,velo,testCurrent);
	END_IF
END_IF


IF testZeroCurrent THEN
	IBDMotor.SetTorque(0);
	testZeroCurrent := FALSE;
END_IF

IF testSomeCurrent THEN
	IBDMotor.SetTorque(testCurrent);
	testSomeCurrent := FALSE;
END_IF


IF resetONS.Q THEN
	IBDMotor.Reset();
	//IBDMotor.Reset();
	
	_reset := FALSE;
	//_openIBD := FALSE;
	_closeIBD := FALSE;
	//_homeNow := FALSE;
	startTest := FALSE;
	testActive := FALSE;
	delayTimer.IN := FALSE;
	state := MotorizedIBDStates.Idle; 
END_IF

IF (IBDMotor.Faulted AND NOT disableFaults)
	AND state <> MotorizedIBDStates.Faulted
THEN
	state := MotorizedIBDStates.Faulting; 
END_IF

homeRequiredONS(CLK := IBDMotor.homeRequired);
IF homeRequiredONS.OSR THEN
	homeRequired := TRUE;
END_IF

_ready := state = MotorizedIBDStates.Idle AND NOT homeRequired AND IBDOpen;

CASE state OF
	MotorizedIBDStates.Idle :					//
										IF startTest THEN
											startTest := FALSE;
											testActive := TRUE;
											IF IBDMotor.homeRequired THEN
												IBDMotor.HomeNow();
												state := MotorizedIBDStates.Homing;
											ELSE
												state := MotorizedIBDStates.Initialize;
											END_IF
												
										END_IF
											
										IF _homeNow THEN
											_homeNow := FALSE;
											//IF IBDMotor.HomeRequired THEN
												IBDMotor.HomeNow();
											//END_IF
											delayTimer.PT := T#150MS;
											delayTimer.IN := TRUE;
											state := MotorizedIBDStates.Homing;
										END_IF
										
										IF _openIBD AND NOT _reset THEN
											
											state := MotorizedIBDStates.MoveJawOut;
										END_IF
										
										IF _closeIBD THEN
											_closeIBD := FALSE;
											state := MotorizedIBDStates.MoveJawIn;
										END_IF
										
										IF _openFull THEN
											_openFull := FALSE;
											state := MotorizedIBDStates.MoveOutFull;
										END_IF
	
	MotorizedIBDStates.Homing :				//
										
										IF NOT (IBDMotor.homeRequired) AND delayTimer.Q THEN
											delayTimer.IN := FALSE;
											homeRequired := FALSE;
											state := MotorizedIBDStates.Initialize;
										END_IF
	
	
	MotorizedIBDStates.Initialize :			//
										
										IF IBDOpen THEN
											state := MotorizedIBDStates.Initialized;
										ELSE
											IBDMotor.MoveToPosition(pbarOutSetting,accel,decel,velo);
											//IBDMotor.MoveToPosition(pbarOutSetting,accel,decel,velo);
											state := MotorizedIBDStates.Initializing;
										END_IF
	
	
	MotorizedIBDStates.Initializing :			//
										IF IBDOpen THEN
											state := MotorizedIBDStates.Initialized;
										END_IF
	
	
	MotorizedIBDStates.Initialized :			//
										state := MotorizedIBDStates.Idle;
	
	
	MotorizedIBDStates.MoveJawOut :			//
										
										//IBDMotor.MoveToPositionTorque(pbarOutSetting,accel,decel,velo,testCurrent);
										IBDMotor.MoveToPosition(pbarOutSetting,accel,decel,velo);
										state := MotorizedIBDStates.MovingJawOut;
										_openIBD := FALSE;
										//IBDMotor.SetPositionLimit(150);
	
	MotorizedIBDStates.MovingJawOut :			//
										IF IBDOpen THEN
											state := MotorizedIBDStates.Idle;
										END_IF
	
	
	MotorizedIBDStates.MovedJawOut :			//
										
	
	MotorizedIBDStates.MoveOutFull :			//
										
										//IBDMotor.MoveToPositionTorque(pbarOutSetting,accel,decel,velo,testCurrent);
										IBDMotor.MoveToPosition(12,accel,decel,velo);
										state := MotorizedIBDStates.MovingOutFull;
										//IBDMotor.SetPositionLimit(150);
	
	MotorizedIBDStates.MovingOutFull :			//
										IF IBDFullyOpen THEN
											state := MotorizedIBDStates.Idle;
										END_IF
	
	
	MotorizedIBDStates.MovedOutFull :			//
	
	MotorizedIBDStates.MoveJawIn :				//
									
										IBDMotor.MoveToPositionTorque(pbarInSetting,accel,decel,velo,testCurrent);
										//IBDMotor.MoveToPosition(0,accel,decel,velo+(TO_INT(TO_REAL(velo)*0.25)));
										state := MotorizedIBDStates.MovingJawIn;
	
	
	MotorizedIBDStates.MovingJawIn : 			//
										IF IBDMotor.alarms.currentFoldback OR IBDMotor.InPosition THEN
											state := MotorizedIBDStates.Clamping;
										END_IF
	
	
	MotorizedIBDStates.MovedJawIn :			//
										state := MotorizedIBDStates.StartClamping;
	
	
	MotorizedIBDStates.StartClamping :			//
										
	
	MotorizedIBDStates.StartedClamping :		//
										
	
	
	MotorizedIBDStates.Clamping :				//
										IF _openIBD THEN
											_openIBD := FALSE;
											state := MotorizedIBDStates.MoveJawOut;
										END_IF
											
										IF _openFull THEN
											_openFull := FALSE;
											state := MotorizedIBDStates.MoveOutFull;
										END_IF
	
	
	MotorizedIBDStates.ReleaseClamp :			//  
										
	
	MotorizedIBDStates.ReleasingClamp :		//
										
	
	MotorizedIBDStates.Faulting :			// 
										Globals.jawMovingIn := FALSE;
										_reset := FALSE;
										_openIBD := FALSE;
										_closeIBD := FALSE;
										_homeNow := FALSE;
										startTest := FALSE;
										testActive := FALSE;
										delayTimer.IN := FALSE;
										//IBDMotor.MoveDistanceTorque(velocity:=100, acceleration := 1, deceleration := 1, distance := 0, current := 0);
										IBDMotor.Disable();
										state := MotorizedIBDStates.Faulted;
	
	MotorizedIBDStates.Faulted :				//
	
END_CASE

SUPER^();

METHOD CloseIBD : BOOL
VAR_INPUT
END_VAR
_closeIBD := TRUE;
END_METHOD

METHOD OpenFull : BOOL
VAR_INPUT
END_VAR
_openFull := TRUE;
END_METHOD

METHOD OpenIBD : BOOL
VAR_INPUT
END_VAR
_openIBD := TRUE;
END_METHOD

METHOD RemovePower : BOOL
VAR_INPUT
END_VAR
state := MotorizedIBDStates.Faulting;
homeRequired := TRUE;
END_METHOD

METHOD HomeNow : BOOL
VAR_INPUT
END_VAR
_homeNow := TRUE;
END_METHOD

END_FUNCTION_BLOCK

// Device/Application/FBs/FB_BaggerHeadRaise
FUNCTION_BLOCK FB_BaggerHeadRaise
VAR_INPUT
	faultIndication : BOOL;
	raiseCommand : BOOL;
	lowerCommand : BOOL;
	raiseLimitSwitch : BOOL;
	lowerLimitSwitch : BOOL;
END_VAR
VAR_OUTPUT
	runMotorOutput : BOOL;
	motorDirectionOutput : BOOL;
END_VAR
VAR
END_VAR

IF NOT faultIndication THEN
	IF (raiseCommand AND NOT raiseLimitSwitch) OR (lowerCommand AND NOT lowerLimitSwitch) THEN
		runMotorOutput := TRUE;
	ELSE
		runMotorOutput := FALSE;
	END_IF
	
	IF (lowerCommand AND NOT lowerLimitSwitch) THEN
		motorDirectionOutput := TRUE;
	ELSE
		motorDirectionOutput := FALSE;
	END_IF
	
ELSE
	runMotorOutput := FALSE;
	motorDirectionOutput := FALSE;
END_IF

END_FUNCTION_BLOCK

// Device/Application/FBs/GetTime
FUNCTION_BLOCK GetTime
VAR_INPUT
END_VAR
VAR_OUTPUT
    currentDateAndTime : DATE_AND_TIME;
    
END_VAR
VAR
    iState                    : INT;
    udiUtcTime             : UDINT;
    udiUtcTimeLocal     : UDINT;
    strTimeDate         : SYSTIMEDATE;
    strTimeDateLocal     : SYSTIMEDATE;
    dtDateTimeUTC        : DATE_AND_TIME;
    timeLeftTime        : TIME;
    timeLeftDWORD        : DWORD;
    dDateUTC            : DATE;
    todTimeOfDayUTC        : TOD;
    
    tSysStartTime        : TIME;
    systimeStartNano    : SYSTIME;
    udiStartTimeResult    : UDINT;
    
    udiResult             : UDINT;
    
    
    GetDateAndTime            : DTU.GetDateAndTime;
    SetTimeZoneInformation    : DTU.SetTimeZoneInformation;
    
    dtCurrent                : DATE_AND_TIME;
    dtConcated                : DATE_AND_TIME;
    eWeekday                 : RTCLK.WEEKDAY;
    uiYear                     : UINT;
    uiMonth                     : UINT;
    uiDay                     : UINT;
    uiHour                     : UINT;
    uiMinute                 : UINT;
    uiSecond                 : UINT;
        
    dtuError                : DTU.ERROR;
END_VAR

CASE iState OF

    0:    
        iState:= 1;
        
    1:  // retrieves the target date and time, including the timezone information which was set before
        GetDateAndTime( xExecute:= TRUE);
        IF GetDateAndTime.xDone THEN
            dtCurrent:= GetDateAndTime.dtDateAndTime;
            GetDateAndTime(xExecute:= FALSE);
			currentDateAndTime := dtCurrent;
            //timeLeft := TIME_TO_DT(DT_TO_TIME(targetDate) - DT_TO_TIME(dttarget));
            iState:= 2;
        END_IF
        IF GetDateAndTime.xError THEN
            GetDateAndTime(xExecute:= FALSE);
            iState:= 32767;
        END_IF
    
    2: (*set a spedific date and time --> returns a variable of type DATE_AND_TIME 
         DateConcat --> set only date information --> returns a variable of type DATE
         TODConcat  --> set only the time information  --> returns a variable of TOD (Time of day) *)
        IF dtuError = 0 THEN
            iState := 3;
        ELSE
            iState := 32767;
        END_IF
        
    3:  (*a DATE_AND_TIME variable is splitted in its parts, like year, month, day etc.
            DateSplit --> the same function for a DATE variable
            TODSplit  --> the same function for a TOD variable *)

            
        IF dtuError = 0 THEN
            iState:= 1;
        ELSE
            iState:= 32767;
        END_IF
        
    32767: ; //error

END_CASE

END_FUNCTION_BLOCK

// Project Information/GetVersion
// This function has been automatically generated from the project information.
{attribute 'signature_flag' := '1073741824'}
{attribute 'register_in_runtime'}
FUNCTION GetVersion : VERSION
VAR_INPUT
	
END_VAR

GetVersion.uiMajor := 0;
GetVersion.uiMinor := 9;
GetVersion.uiServicePack := 13;
GetVersion.uiPatch := 2;

END_FUNCTION

// Project Information/GetTextProperty
// This function has been automatically generated from the project information.
{attribute 'signature_flag' := '1073741824'}
{attribute 'register_in_runtime'}
FUNCTION GetTextProperty : WSTRING
VAR_INPUT
	stKey: WSTRING;
END_VAR

IF stKey = "Author" THEN
	GetTextProperty := "Ben Hess";
ELSIF stKey = "Company" THEN
	GetTextProperty := "Sharp Packaging";
ELSIF stKey = "Project" THEN
	GetTextProperty := "AlphaController";
ELSIF stKey = "Title" THEN
	GetTextProperty := "MOAB Prototype";
ELSIF stKey = "VersionPostfix" THEN
	GetTextProperty := "-alpha/pro24";
ELSE
	GetTextProperty := "";
END_IF

END_FUNCTION

// Device/Application/Event Handlers/StartDone
FUNCTION StartDone : DWORD
VAR_IN_OUT
	EventPrm: CmpApp.EVTPARAM_CmpApp;
END_VAR
VAR
END_VAR

Globals.firstScan := TRUE;
RecallValues();

END_FUNCTION

// Device/Application/FBs/TimeLeftFB
FUNCTION_BLOCK TimeLeftFB
VAR_INPUT
    targetDate : DATE_AND_TIME;
END_VAR
VAR_OUTPUT
    timeLeft : DATE_AND_TIME;
    
    targetMonths : UINT;
    targetDays : UINT;
    targetHours : UINT;
    targetMinutes : UINT;
    targetSeconds : UINT;
    currentMonths : UINT;
    currentDays : UINT;
    currentHours : UINT;
    currentMinutes : UINT;
    currentSeconds : UINT;
    timeLeftMonths : UINT;
    timeLeftDays : UINT;
    timeLeftHours : UINT;
    timeLeftMinutes : UINT;
    timeLeftSeconds : UINT;
    timeLeftString : STRING[250];
END_VAR
VAR
    iState                    : INT;
    udiUtcTime             : UDINT;
    udiUtcTimeLocal     : UDINT;
    strTimeDate         : SYSTIMEDATE;
    strTimeDateLocal     : SYSTIMEDATE;
    dtDateTimeUTC        : DATE_AND_TIME;
    timeLeftTime        : TIME;
    timeLeftDWORD        : DWORD;
    dDateUTC            : DATE;
    todTimeOfDayUTC        : TOD;
    
    tSysStartTime        : TIME;
    systimeStartNano    : SYSTIME;
    udiStartTimeResult    : UDINT;
    
    udiResult             : UDINT;
    
    
    GetDateAndTime            : DTU.GetDateAndTime;
    SetTimeZoneInformation    : DTU.SetTimeZoneInformation;
    
    dtCurrent                : DATE_AND_TIME;
    dtConcated                : DATE_AND_TIME;
    eWeekday                 : RTCLK.WEEKDAY;
    uiYear                     : UINT;
    uiMonth                     : UINT;
    uiDay                     : UINT;
    uiHour                     : UINT;
    uiMinute                 : UINT;
    uiSecond                 : UINT;
        
    dtuError                : DTU.ERROR;
END_VAR

CASE iState OF

    0:    
        iState:= 1;
        
    1:  // retrieves the target date and time, including the timezone information which was set before
        GetDateAndTime( xExecute:= TRUE);
        IF GetDateAndTime.xDone THEN
            dtCurrent:= GetDateAndTime.dtDateAndTime;
            GetDateAndTime(xExecute:= FALSE);
            //timeLeft := TIME_TO_DT(DT_TO_TIME(targetDate) - DT_TO_TIME(dttarget));
            iState:= 2;
        END_IF
        IF GetDateAndTime.xError THEN
            GetDateAndTime(xExecute:= FALSE);
            iState:= 32767;
        END_IF
    
    2: (*set a spedific date and time --> returns a variable of type DATE_AND_TIME 
         DateConcat --> set only date information --> returns a variable of type DATE
         TODConcat  --> set only the time information  --> returns a variable of TOD (Time of day) *)
        dtConcated := DTU.DTConcat(uiYear:= 2010, uiMonth:= 10, uiDay:= 5, 
                            uiHour:= 9, uiMinute:= 20, uiSecond:= 12, peError:=ADR(dtuError));
        IF dtuError = 0 THEN
            iState := 3;
        ELSE
            iState := 32767;
        END_IF
        
    3:  (*a DATE_AND_TIME variable is splitted in its parts, like year, month, day etc.
            DateSplit --> the same function for a DATE variable
            TODSplit  --> the same function for a TOD variable *)
        dtuError := DTU.DTSplit(
            dtDateAndTime := dtCurrent,
            puiYear := ADR(uiYear), 
            puiMonth := ADR(currentMonths), 
            puiDay := ADR(currentDays), 
            puiHour := ADR(currentHours), 
            puiMinute := ADR(currentMinutes), 
            puiSecond := ADR(currentSeconds));
        dtuError := DTU.DTSplit(
            dtDateAndTime := targetDate,
            puiYear := ADR(uiYear), 
            puiMonth := ADR(targetMonths), 
            puiDay := ADR(targetDays), 
            puiHour := ADR(targetHours), 
            puiMinute := ADR(targetMinutes), 
            puiSecond := ADR(targetSeconds));
            
        IF dtuError = 0 THEN
            iState:= 1;
        ELSE
            iState:= 32767;
        END_IF
        
    32767: ; //error

END_CASE

timeLeftMonths := currentMonths - targetMonths;
timeLeftDays := currentDays - targetDays;
timeLeftHours := currentHours - targetHours;
timeLeftMinutes := currentMinutes - targetMinutes;
timeLeftSeconds := currentSeconds - targetSeconds;

timeLeftString := CONCAT('Time left to PMMI: ', UINT_TO_STRING(timeLeftMonths));
timeLeftString := CONCAT(' Months, ', UINT_TO_STRING(timeLeftDays));
timeLeftString := CONCAT(' Days, ', UINT_TO_STRING(timeLeftHours));
timeLeftString := CONCAT(' Hours, ', UINT_TO_STRING(timeLeftMinutes));
timeLeftString := CONCAT(' Minutes, ', UINT_TO_STRING(timeLeftSeconds));
timeLeftString := CONCAT(' Seconds', '');

timeLeftDWORD := DT_TO_DWORD(targetDate) - DT_TO_DWORD(dtCurrent);
timeLeftDays := DWORD_TO_UINT(timeLeftDWORD / 86000);

END_FUNCTION_BLOCK

// Device/Application/FBs/FB_WriteToFile
FUNCTION_BLOCK FB_WriteToFile
VAR_INPUT
   xFilePath: STRING;
   xText_Write: STRING(2000);
   xAppend_OverWrite: BOOL;
   xAppend_Pos: UDINT;
   xWrite: BOOL;
   xRead: BOOL;
   xLine_No_To_Read: UDINT;   
END_VAR
VAR_OUTPUT
   xText_Read: STRING(2000);
   xDone: BOOL;
END_VAR
VAR
   
// Write Variables
   xWrite_Trig: R_TRIG;
   xStart_Write: BOOL;
   xNew_Line: STRING(2000);
   
// Read Variables
   xRead_Trig: R_TRIG;
   xStart_Read: BOOL;
   xLine_Read: UDINT;
   
   hFile           : RTS_IEC_HANDLE := RTS_INVALID_HANDLE;
   udiBytesRead    : UDINT;
   udiBytesCopied   : UDINT;
   udiWrite      : UDINT;
   udiFileSize     : UDINT;
   udiPos         : UDINT;

//(* Error Codes *)
   udiPosError          : RTS_IEC_RESULT;
   udiCopyError      : RTS_IEC_RESULT;
   udiDeleteError1      : RTS_IEC_RESULT;
   udiDeleteError2      : RTS_IEC_RESULT;
   udiWriteError1      : RTS_IEC_RESULT;
   udiWriteError2      : RTS_IEC_RESULT;
   udiWriteError3      : RTS_IEC_RESULT;
   udiOpenError1      : RTS_IEC_RESULT;
   udiOpenError2      : RTS_IEC_RESULT;
   udiOpenError3      : RTS_IEC_RESULT;
   udiOpenError4      : RTS_IEC_RESULT;

   udiReadError1   : RTS_IEC_RESULT;
   udiReadError2   : RTS_IEC_RESULT;
   udiReadError3   : RTS_IEC_RESULT;
   udiCloseError1   : RTS_IEC_RESULT;
   udiCloseError2   : RTS_IEC_RESULT;
   udiCloseError3   : RTS_IEC_RESULT;
   udiCloseError4   : RTS_IEC_RESULT;
   udiSizeError : RTS_IEC_RESULT;
   udiDirDeleteError: UDINT; 
   udiCreateError: UDINT;
END_VAR

xWrite_Trig();
//xWrite_Trig.PT:= T#500MS;
xWrite_Trig.CLK:= xWrite;
xStart_Write:= xWrite_Trig.Q;

xRead_Trig();
//xRead_Trig.PT:= T#500MS;
xRead_Trig.CLK:= xRead;
xStart_Read:= xRead_Trig.Q;

IF xStart_Write THEN
   xDone:= FALSE;
   IF xAppend_OverWrite THEN 
   hFile:= SysFileOpen(szFile:= xFilePath, am:= ACCESS_MODE.AM_APPEND, pResult:= ADR(udiOpenError1));
   END_IF
   IF xAppend_OverWrite = FALSE THEN
      hFile:= SysFileOpen(szFile:= xFilePath, am:= ACCESS_MODE.AM_WRITE_PLUS, pResult:= ADR(udiOpenError1));
   END_IF
   udiPosError:= SysFileGetPos(hFile:= hFile, pulPos:= ADR(udiPos));
   IF hFile <> RTS_INVALID_HANDLE THEN
      xNew_Line:= concat('$n', xText_Write);
      IF udiPos = 16#0 THEN
         udiWrite:= SysFileWrite(hFile:= hFile, pbyBuffer:= ADR(xText_Write), ulSize:= INT_TO_UDINT(LEN(xText_Write)), pResult:= ADR(udiWriteError1));
      ELSE
         udiWrite:= SysFileWrite(hFile:= hFile, pbyBuffer:= ADR(xNew_Line), ulSize:= INT_TO_UDINT(LEN(xNew_Line)), pResult:= ADR(udiWriteError1));
      END_IF
      udiCloseError1:= SysFileClose(hFile:= hFile);
   END_IF
   xDone:= TRUE;
END_IF

IF xStart_Read THEN
   xDone:= FALSE;
   hFile:= SysFileOpen(szFile:= xFilePath, am:= ACCESS_MODE.AM_READ, pResult:= ADR(udiOpenError1));
   IF hFile <> RTS_INVALID_HANDLE THEN
      udiBytesRead := SysFileRead(hFile:= hFile, pbyBuffer:= ADR(xText_Read), ulSize:=SIZEOF(xText_Read), pResult:=ADR(udiReadError1));
      xText_Read[udiBytesRead]:= 0;
   END_IF
   //xDone:= TRUE;   
END_IF

END_FUNCTION_BLOCK

// Device/Application/FBs/Cylinders/FB_CylinderWithFeedback
FUNCTION_BLOCK FB_CylinderWithFeedback EXTENDS FB_Cylinder IMPLEMENTS ICylinder, IFault
VAR_INPUT
    extendedFeedbackInput : BOOL;    //Extended feedback input from I/O
    retractedFeedbackInput : BOOL;    //Retracted feedback input from I/O
    extendFaultDelay : INT := 1000;        //Extend fault delay in MS
    retractFaultDelay : INT := 1000;        //Retract fault delay in MS
    faultMonitoring : BOOL;                    //Fault monitoring enabled if true
END_VAR
VAR_OUTPUT
    failedToExtend : FB_Fault;            //Failed to Extend Fault
    failedToRetract : FB_Fault;            //Failed to Retract Fault
END_VAR
VAR
    faultIndication : BOOL;            //Overall fault status of cylinder
    extendFaultTimer : TON;            //Extend Fault Timer
    retractFaultTimer : TON;        //Retract Fault Timer
    resetFaults : BOOL;                //Reset faults
END_VAR

METHOD Execute
//This code monitors the positon of the cylinder and raises a fault if the cylinder doesn't reach its
//desired postion within the specified time.

//Initialize timers
extendFaultTimer(PT := INT_TO_TIME(extendFaultDelay));
retractFaultTimer(PT := INT_TO_TIME(retractFaultDelay));

//Only enable timers if we are to be monitoring faults
IF faultMonitoring THEN
    extendFaultTimer.IN := (extendOutput AND NOT extendedFeedbackInput);
    retractFaultTimer.IN := (retractOutput AND NOT retractedFeedbackInput);
ELSE 
        extendFaultTimer.IN := FALSE;
        retractFaultTimer.IN := FALSE;
END_IF

//Rasie the alarms
failedToExtend.faultTrigger := extendFaultTimer.Q;
failedToRetract.faultTrigger := retractFaultTimer.Q;

//Set overall fault indication
//faultIndication := failedToExtend.Active OR failedToRetract;
END_METHOD

END_FUNCTION_BLOCK

// Device/Application/FBs/Fault/FB_GetTime
FUNCTION_BLOCK FB_GetTime
VAR_INPUT
END_VAR
VAR_OUTPUT
    currentDateAndTime : DATE_AND_TIME;
    
END_VAR
VAR
    iState                    : INT;
    udiUtcTime             : UDINT;
    udiUtcTimeLocal     : UDINT;
    strTimeDate         : SYSTIMEDATE;
    strTimeDateLocal     : SYSTIMEDATE;
    dtDateTimeUTC        : DATE_AND_TIME;
    timeLeftTime        : TIME;
    timeLeftDWORD        : DWORD;
    dDateUTC            : DATE;
    todTimeOfDayUTC        : TOD;
    
    tSysStartTime        : TIME;
    systimeStartNano    : SYSTIME;
    udiStartTimeResult    : UDINT;
    
    udiResult             : UDINT;
    
    
    GetDateAndTime            : DTU.GetDateAndTime;
    SetTimeZoneInformation    : DTU.SetTimeZoneInformation;
    
    dtCurrent                : DATE_AND_TIME;
    dtConcated                : DATE_AND_TIME;
    eWeekday                 : RTCLK.WEEKDAY;
    uiYear                     : UINT;
    uiMonth                     : UINT;
    uiDay                     : UINT;
    uiHour                     : UINT;
    uiMinute                 : UINT;
    uiSecond                 : UINT;
        
    dtuError                : DTU.ERROR;
END_VAR

CASE iState OF

    0:    
        iState:= 1;
        
    1:  // retrieves the target date and time, including the timezone information which was set before
        GetDateAndTime( xExecute:= TRUE);
        IF GetDateAndTime.xDone THEN
            dtCurrent:= GetDateAndTime.dtDateAndTime;
            GetDateAndTime(xExecute:= FALSE);
			currentDateAndTime := dtCurrent;
            //timeLeft := TIME_TO_DT(DT_TO_TIME(targetDate) - DT_TO_TIME(dttarget));
            iState:= 2;
        END_IF
        IF GetDateAndTime.xError THEN
            GetDateAndTime(xExecute:= FALSE);
            iState:= 32767;
        END_IF
    
    2: (*set a spedific date and time --> returns a variable of type DATE_AND_TIME 
         DateConcat --> set only date information --> returns a variable of type DATE
         TODConcat  --> set only the time information  --> returns a variable of TOD (Time of day) *)
        IF dtuError = 0 THEN
            iState := 3;
        ELSE
            iState := 32767;
        END_IF
        
    3:  (*a DATE_AND_TIME variable is splitted in its parts, like year, month, day etc.
            DateSplit --> the same function for a DATE variable
            TODSplit  --> the same function for a TOD variable *)

            
        IF dtuError = 0 THEN
            iState:= 1;
        ELSE
            iState:= 32767;
        END_IF
        
    32767: ; //error

END_CASE

END_FUNCTION_BLOCK

// Device/Application/ObjectHandling/FB_CollectionHandlerAll
FUNCTION_BLOCK FINAL FB_CollectionHandlerAll
VAR_INPUT
END_VAR
VAR
	Collection: ARRAY[0..GlobalObjects.MAX_OBJECTS] OF IAllObjects; // object array
	ObjNames   : ARRAY[0..GlobalObjects.MAX_OBJECTS] OF STRING;
	_ArrayOver   : BOOL;
	_BadObj      : INT;
	_DupeObj   : INT;
	_OverObj   : INT;
	_TotalObj   : UINT;
END_VAR

METHOD FINAL AddObject
VAR_INPUT
	Obj   : IAllObjects;
END_VAR
VAR
	AnyObject : IAllObjects;
	Fault : IFault;
	Cylinder : ICylinder;
	PositionableMotor : IPositionableMotor;
	Logger : IMachineLogger;
	Loggable : ILoggable;
	Executable : IExecuteAutomatically;
	Initializable : IInitializable;
	J   : UINT;
END_VAR
IF (__QUERYINTERFACE(Obj, AnyObject)) THEN
   // make sure haven't already added this object
   FOR J:= 1 TO _TotalObj DO
      IF Collection[J] = AnyObject THEN
         // object pointer matches - dupe!
         _DupeObj:= _DupeObj + 1;
         RETURN;
      END_IF
   END_FOR
   
   IF _TotalObj < GlobalObjects.MAX_OBJECTS THEN
      Collection[_TotalObj]:= AnyObject;
      ObjNames[_TotalObj]:= Obj.InstanceName;
	   _TotalObj:= _TotalObj + 1;
   ELSE
      _ArrayOver:= TRUE;
      _OverObj:= _OverObj + 1;
   END_IF
ELSE
   _BadObj:= _BadObj + 1;
END_IF

// Add object to proper collection based on its interfaces
IF (__QUERYINTERFACE(Obj, Fault)) THEN
	GlobalObjects.CollectionOfFaults.AddObject(Fault);
END_IF

// IF (__QUERYINTERFACE(Obj, Cylinder)) THEN
// 	GlobalObjects.CollectionOfCylinders.AddObject(Cylinder);
// END_IF
// 
// IF (__QUERYINTERFACE(Obj, PositionableMotor)) THEN
// 	GlobalObjects.CollectionOfPositionableMotors.AddObject(PositionableMotor);
// END_IF

IF (__QUERYINTERFACE(Obj, Logger)) THEN
	GlobalObjects.CollectionOfLogs.AddObject(Logger);
END_IF

IF (__QUERYINTERFACE(Obj, Loggable)) THEN
	GlobalObjects.CollectionOfLoggable.AddObject(Loggable);
END_IF

IF (__QUERYINTERFACE(Obj, Executable)) THEN
	GlobalObjects.CollectionOfExecutable.AddObject(Executable);
END_IF

IF (__QUERYINTERFACE(Obj, Initializable)) THEN
	GlobalObjects.CollectionOfInitialzable.AddObject(Initializable);
END_IF
END_METHOD

END_FUNCTION_BLOCK

// Device/Application/FBs/Components/BagDeliveryFB_BothMotors
FUNCTION_BLOCK BagDeliveryFB_BothMotors EXTENDS BaseComponentFB IMPLEMENTS IComponentStatus
VAR_INPUT
    feedBagPB : BOOL;                // Manually Feed bag out
	jogForwardPB : BOOL;
	jogReversePB : BOOL;
    bagsToFeedSetpoint : INT;        // Bags to feed setpoint for testing
    reverseDistanceSetpoint : REAL := -3;  // Distance to reverse
    bagLengthSetpoint : REAL := 23.5;  // Bag length to feed
    accelSetpoint : INT := 600;            // Acceleration Setpoint
    decelSetpoint : INT := 2000;        // Deceleration Setpoint
    reverseVelocitySetpoint : INT := 3;            // Reverse Velocity setoint (IPS)
    feedVelocitySetpoint : INT := 55;            // Bag Feed Velocity setoint (IPS)
    printVelocitySetpoint : UDINT := 6;            // Print speed (IPS)
    sealOffsetSetpoint : REAL := 1.5;            // Seal Offset
    printOffsetSetpoint : REAL := 3;            // Print Offset
    printLengthSetpoint : REAL := 8;                    // Print length
	reverseToPrintHeadSetpoint : REAL := -1.25;
	feedToPhotoeyeSetpoint : REAL := 2.0;
	useLastPrinterDelta : BOOL := TRUE;
	tensionFailONS : FB_ONS;
END_VAR
VAR_OUTPUT
    state : BAG_DELIVERY_STATES;    // Current state of bag delivery component
	reverseFault : FB_Fault(name := 'Reverse Fault');
	noBagOverEye : FB_Fault(name := 'No bag over Photoeye');
	bagTensionFault : FB_Fault(name := 'Bag Tension Fault');
END_VAR
VAR
    delay : TON := (PT := T#100MS);    // Delay for testing
	jogForwardONS: FB_ONS;
	jogReverseONS: FB_ONS;
	delayForReverseFault : Standard.TON;
	autoFeedDelay : TON := (PT := T#200MS);
	sealBarToPrintHeadLength : REAL;
    bagsCurrentlyFed  :INT;            // Bags currently fed for testing
    remainingLength : REAL;            // Remaining bag length after print
	delayForPrintFeed : TIME := T#250MS;
	printerExtraFeedLength : REAL := 0.25;
    //bagFeedMasterMotor : FB_AppliedMotionStepServoTCP();
    //bagFeedMasterMotor : FB_AppliedMotionBagDeliveryMotor();
	bagFeedMasterMotor : FB_AppliedMotionBagDeliveryMotor_1();
	//bagFeedRearMotor : FB_AppliedMotionBagDeliveryMotor_1();
	bagFeedRearMotor : FB_AppliedMotionStepServoEIPBase();
	accelPercent : REAL := 0.1;
	decelPercent : REAL := 0.05;
    _amReverseBag : BOOL;            // Auto Mode - Reverse bag
    _amFeedBagOut : BOOL;            // Auto Mode - Feed new bag out
    _amWaitForPrinter : BOOL;        // Auto Mode - wait for printer
    _amPrinterReady : BOOL;            // Auto Mode - Printer is ready
    _amStartPrint : BOOL;            // Auto Mode - Start Printing
    _amPrinterDone : BOOL;             // Auto Mode - Printer is Done
	_amFeedToEye : BOOL;			  // Auto Mode - Feed Bag to Eye
END_VAR

//    Function Block: BagDeliveryFB
//    Description: This is the state machine for the bag delivery test rig
//    
//    Created by: Ben Hess
//    Created Date: Thursday, April 19, 2018

SUPER^();
tensionFailONS(CLK := iBagTensionFault);

delay();
delayForReverseFault();
autoFeedDelay(IN := _amFeedBagOut);
// This is the master Applied Motion motor
IF useLastPrinterDelta THEN
	IF Globals.lastPrinterDelta >= T#90MS THEN
		delayForPrintFeed := Globals.lastPrinterDelta - T#80MS;
	ELSE
		delayForPrintFeed := T#10MS;
	END_IF
END_IF
bagLengthSetpoint := HMIData.bagLength;
printVelocitySetpoint := HMIData.printSpeed;
sealOffsetSetpoint := HMIData.bagSkirtLength;
printOffsetSetpoint := HMIData.printOffset;
sealBarToPrintHeadLength := ABS(reverseToPrintHeadSetpoint) + 2.25;
printLengthSetpoint := HMIData.printLength;
reverseVelocitySetpoint := TO_INT(HMIData.bagReverseSpeed);
feedVelocitySetpoint := TO_INT(HMIData.bagForwardSpeed);

(*bagFeedMasterMotor(modbusInputParameters := BagDeliverMasterMotorModbusInputs, 
                    stepsPerInchSetpoint := Globals.STEPS_PER_INCH_20_DEGREE_BAG_DELIVERY, 
                    reversePolarity := FALSE, 
                    slave := Bag_Delivery_Master_Motor);*)
bagFeedMasterMotor(ptrEIPInputs := ADR(bagDeliveryMotorInputs),
                ptrEIPOutputs := ADR(bagDeliveryMotorOutputs),
                stepsPerInchSetpoint := Globals.STEPS_PER_INCH_20_DEGREE_BAG_DELIVERY,
                //faultHandler := PRG_Bagger.faultHandler,
				reversePolarity := FALSE, 
				defaultCurrentSetpoint := 1150, 
				commFail := Bag_Delivery_EIP_Motor.udiState <> 4);
bagFeedMasterMotor.Execute();

bagFeedRearMotor(ptrEIPInputs := ADR(bagRearMotorInputs),
                ptrEIPOutputs := ADR(bagRearMotorOutputs),
                stepsPerInchSetpoint := Globals.STEPS_PER_INCH_20_DEGREE_BAG_DELIVERY,
                //faultHandler := PRG_Bagger.faultHandler,
				reversePolarity := FALSE, 
				defaultCurrentSetpoint := 1150, 
				commFail := Bag_Delivery_Rear_Motor.udiState <> 4);
bagFeedRearMotor.Execute();

IF enableONS.Q OR resetONS.Q THEN
    IF _mode = DEVICE_MODES.Manual THEN 
        state := BAG_DELIVERY_STATES.Manual;
    ELSE
        state := BAG_DELIVERY_STATES.Idle;
    END_IF
	_reset := FALSE;
	ClearCommands();
END_IF
jogForwardONS(CLK := jogForwardPB);
jogReverseONS(CLK := jogReversePB);
IF NOT enable THEN
    state := BAG_DELIVERY_STATES.Idle;
END_IF
delay();
_ready := (_mode = DEVICE_MODES.Auto) AND (NOT (state = BAG_DELIVERY_STATES.Fault) OR NOT (state = BAG_DELIVERY_STATES.Idle));

IF tensionFailONS.OSR THEN
	bagTensionFault.Trigger();
END_IF

